(* CoDeSys 2.3.9.41 project: rePlc160.pro *)
(* Libraries: STANDARD.LIB 4.10.05 10:14:46, SmsOwenLib.lib 5.10.12 16:48:36, IECSFC.LIB 13.4.06 14:51:28, Util.lib 18.5.10 15:14:28, SysLibCom.lib 20.2.06 13:31:08, UNM.lib 14.2.06 12:27:08, SMS.lib 29.7.11 08:51:48, SYSLIBTIME.LIB 20.2.06 13:31:16, SYSTASKINFO.LIB 20.2.06 13:31:38, ANALYZATION.LIB 5.10.99 08:05:06, SYSLIBCALLBACK.LIB 20.2.06 13:31:08 *)

(* PLC configuration (modules and I/O channels)
Fast discrete inputs [I_SIMPLE_INPUT] node 0, in %IB0 out %QB0 {Filtrationtime = 10}
  DI_leakSens1 AT %IX0.0 [BitInput] Discrete input 1
  DI_leakSens2 AT %IX0.1 [BitInput] Discrete input 2
  DI_lamp1 AT %IX0.2 [BitInput] Discrete input 3
  DI_lamp2 AT %IX0.3 [BitInput] Discrete input 4
Discrete inputs [ID130] node 1, in %IB1 out %QB1 {Filtrationtime_GeneralINP = 10; Visibility = No; PinCount = 12}
  AT %IB1.0 [ByteInput] DI_POLIW
  AT %IB1.1 [ByteInput] DI_FOUNTAIN
Discrete outputs [ID131] node 2, in %IB2 out %QB2 {SafeValueByte = 0; SafeValueByteM = 0; Visibility = No; PinCount = 12}
  AT %QB2.0 [ByteOutput] DO_POLIW_FOUN_LEAK
  AT %QB2.1 [ByteOutput] DO_FOUN
Fast analog inputs [ID125] node 3, in %IB3 out %QB3 {Flt_Comm = 50Hz 2Por}
  AI_01 AT %IR3.0 [FloatInputP] AI #1 {AIN_TYPE = 0-20 mA; Peak_Filtr = 200; Flt_Ch = Off; TauRC = 10; MinFV = 0; MaxFV = 20000.0}
  AI_02 AT %IR3.1 [FloatInputP] AI #2 {AIN_TYPE = 0-20 mA; Peak_Filtr = 200; Flt_Ch = Off; TauRC = 10; MinFV = 0; MaxFV = 20000.0}
  AI_03 AT %IR3.2 [FloatInputP] AI #3 {AIN_TYPE = 0-20 mA; Peak_Filtr = 200; Flt_Ch = Off; TauRC = 10; MinFV = 0; MaxFV = 20000.0}
  AI_04 AT %IR3.3 [FloatInputP] AI #4 {AIN_TYPE = 0-20 mA; Peak_Filtr = 200; Flt_Ch = Off; TauRC = 10; MinFV = 0; MaxFV = 20000.0}
  AI_05 AT %IR3.4 [FloatInputP] AI #5 {AIN_TYPE = 0-20 mA; Peak_Filtr = 200; Flt_Ch = Off; TauRC = 10; MinFV = 0; MaxFV = 20000.0}
  AI_06 AT %IR3.5 [FloatInputP] AI #6 {AIN_TYPE = 0-20 mA; Peak_Filtr = 200; Flt_Ch = Off; TauRC = 10; MinFV = 0; MaxFV = 20000.0}
  AI_07 AT %IR3.6 [FloatInputP] AI #7 {AIN_TYPE = 0-20 mA; Peak_Filtr = 200; Flt_Ch = Off; TauRC = 10; MinFV = 0; MaxFV = 20000.0}
  AI_08 AT %IR3.7 [FloatInputP] AI #8 {AIN_TYPE = 0-20 mA; Peak_Filtr = 200; Flt_Ch = Off; TauRC = 10; MinFV = 0; MaxFV = 20000.0}
  AT %IW3.8 [WordInput] AI read time (10ms)
Analog outputs [ID126] node 4, in %IB4 out %QB4
  AO_fc AT %QR4.0 [FloatOutputP] AO #1 {AOUT_TYPE = 0-10V; SafeValueREAL = 0.0}
  AO_dim1 AT %QR4.1 [FloatOutputP] AO #2 {AOUT_TYPE = 0-10V; SafeValueREAL = 0.0}
  AO_dim2 AT %QR4.2 [FloatOutputP] AO #3 {AOUT_TYPE = 0-10V; SafeValueREAL = 0.0}
  AO_dim3 AT %QR4.3 [FloatOutputP] AO #4 {AOUT_TYPE = 0-10V; SafeValueREAL = 0.0}
Special input [ID103] node 5, in %IB5 out %QB5 {Filtrationtime = 1000; PinCount = 1; WatchDogPeriod = 400; PollPeriod = 3000; Visibility = No}
  AT %IX5.0 [BitInput] Special input
Special output [ID104] node 6, in %IB6 out %QB6 {Visibility = No; PinCount = 1}
  AT %QX6.0 [BitOutput] Special output
Universal network module [UNM_ID300] node 7, in %IB7 out %QB7 {Visibility = No}
  RS-232 [COM2_USART] node 0, in %IB7.0 out %QB7.0 {CommunicationSpeed = 9600; Parity = NO PARITY CHECK; BitLength = 8 bits; StopLength = One stop bit; InterfaceType = RS232; FrameOriented = ASCII; Timeout = 0; Visibility = No}
AT %QD8.0 [DWordOutput] Last address
AT %QW8.1 [WordOutput] Last error
AT %QB8.0.0 [ByteOutput] Line Status
AT %QB8.0.1 [ByteOutput] Modem Fault
AT %QB8.0.2 [ByteOutput] Start_Auto_Dial
AT %QB8.0.3 [ByteOutput] Stop_Dial
RS-232 [COM2_USART] node 0, in %IB8.0.0 out %QB8.0.0 {CommunicationSpeed = 9600; Parity = NO PARITY CHECK; BitLength = 8 bits; StopLength = One stop bit; InterfaceType = RS232; FrameOriented = ASCII; Timeout = 0; Visibility = No}
PPP_Driver [PPP] node 1, in %IB8.0.1 out %QB8.0.1 {LoginString = mts; PasswordString = mts}
Universal Modbus device [ID2000] node 1, in %IB8.1 out %QB8.1 {ModuleIP = 10:10:122:200; ServiceTimeout = 150; TCPport = 502; NetMode = TCP; ModuleSlaveAddress = 1; RequestType = By command; PeriodOfService = 1000; Visibility = No; RepeatCounter = 0; ByteSequence = Trace_mode}
  AT %QB8.1.0 [ComChannel] Command (0xff - Start)
pad_PoliwDIST AT %IW8.1.0.0 [WordInput]
pad_PoliwTELE AT %QW8.1.1.0 [WordOutput]
Register input module [ID2003] node 2, in %IB8.1.2 out %QB8.1.2 {ModbusAddress = 0; Command_read_regs = Read holding Registers  (0x03); Visibility = No}
  FounDIST AT %IW8.1.2.0 [WordInput]
Register output module [ID2004] node 3, in %IB8.1.3 out %QB8.1.3 {ModbusAddress = 0; Command_write_one_reg = Preset singl register (0x06); Visibility = No}
  FounTELE AT %QW8.1.3.0 [WordOutput]
Register output module [ID2004] node 4, in %IB8.1.4 out %QB8.1.4 {ModbusAddress = 0; Command_write_one_reg = Preset singl register (0x06); Visibility = No}
  TRMOUTS AT %QW8.1.4.0 [WordOutput]
AT %QB8.2.0 [ComChannel] Command (0xff - Start)
pad_Voltage AT %QW8.2.0.0 [WordOutput]
pad_Power_A AT %QW8.2.1.0 [WordOutput]
pad_Power_B AT %QW8.2.2.0 [WordOutput]
pad_Power_C AT %QW8.2.3.0 [WordOutput]
pad_Energy AT %QW8.2.4.0 [WordOutput]
pad_trm1_ch1 AT %QW8.2.5.0 [WordOutput]
pad_trm1_ch2 AT %QW8.2.6.0 [WordOutput]
pad_trm1_set1 AT %QW8.2.7.0 [WordOutput]
pad_trm1_set2 AT %QW8.2.8.0 [WordOutput]
pad_trm2_ch1 AT %QW8.2.9.0 [WordOutput]
pad_trm2_ch2 AT %QW8.2.10.0 [WordOutput]
Register output module [ID2004] node 11, in %IB8.2.11 out %QB8.2.11 {ModbusAddress = 11; Command_write_one_reg = Preset singl register (0x06); Visibility = No}
  pad_trm2_set1 AT %QW8.2.11.0 [WordOutput]
Register output module [ID2004] node 12, in %IB8.2.12 out %QB8.2.12 {ModbusAddress = 12; Command_write_one_reg = Preset singl register (0x06); Visibility = No}
  pad_trm2_set2 AT %QW8.2.12.0 [WordOutput]
Universal Modbus device [ID2000] node 3, in %IB8.3 out %QB8.3 {ModuleIP = 10:10:122:200; ServiceTimeout = 150; TCPport = 502; NetMode = TCP; ModuleSlaveAddress = 1; RequestType = By command; PeriodOfService = 7000; Visibility = No; RepeatCounter = 0; ByteSequence = Trace_mode}
  AT %QB8.3.0 [ComChannel] Command (0xff - Start)
  Register input module [ID2003] node 0, in %IB8.3.0 out %QB8.3.0 {ModbusAddress = 0; Command_read_regs = Read holding Registers  (0x03); Visibility = No}
    cir1On AT %IW8.3.0.0 [WordInput]
  Register input module [ID2003] node 1, in %IB8.3.1 out %QB8.3.1 {ModbusAddress = 0; Command_read_regs = Read holding Registers  (0x03); Visibility = No}
    cir1Off AT %IW8.3.1.0 [WordInput]
  Register input module [ID2003] node 2, in %IB8.3.2 out %QB8.3.2 {ModbusAddress = 0; Command_read_regs = Read holding Registers  (0x03); Visibility = No}
    cir2On AT %IW8.3.2.0 [WordInput]
  Register input module [ID2003] node 3, in %IB8.3.3 out %QB8.3.3 {ModbusAddress = 0; Command_read_regs = Read holding Registers  (0x03); Visibility = No}
    cir2Off AT %IW8.3.3.0 [WordInput]
  Register input module [ID2003] node 4, in %IB8.3.4 out %QB8.3.4 {ModbusAddress = 0; Command_read_regs = Read holding Registers  (0x03); Visibility = No}
    cir3On AT %IW8.3.4.0 [WordInput]
  Register input module [ID2003] node 5, in %IB8.3.5 out %QB8.3.5 {ModbusAddress = 0; Command_read_regs = Read holding Registers  (0x03); Visibility = No}
    cir3Off AT %IW8.3.5.0 [WordInput]
  Register input module [ID2003] node 6, in %IB8.3.6 out %QB8.3.6 {ModbusAddress = 0; Command_read_regs = Read holding Registers  (0x03); Visibility = No}
    dist_staticFValue AT %IW8.3.6.0 [WordInput]
  Register input module [ID2003] node 7, in %IB8.3.7 out %QB8.3.7 {ModbusAddress = 0; Command_read_regs = Read holding Registers  (0x03); Visibility = No}
    p1 AT %IW8.3.7.0 [WordInput]
  Register input module [ID2003] node 8, in %IB8.3.8 out %QB8.3.8 {ModbusAddress = 0; Command_read_regs = Read holding Registers  (0x03); Visibility = No}
    p2 AT %IW8.3.8.0 [WordInput]
  Register input module [ID2003] node 9, in %IB8.3.9 out %QB8.3.9 {ModbusAddress = 0; Command_read_regs = Read holding Registers  (0x03); Visibility = No}
    p3 AT %IW8.3.9.0 [WordInput]
  Register input module [ID2003] node 10, in %IB8.3.10 out %QB8.3.10 {ModbusAddress = 0; Command_read_regs = Read holding Registers  (0x03); Visibility = No}
    p4 AT %IW8.3.10.0 [WordInput]
  Register input module [ID2003] node 11, in %IB8.3.11 out %QB8.3.11 {ModbusAddress = 0; Command_read_regs = Read holding Registers  (0x03); Visibility = No}
    p5 AT %IW8.3.11.0 [WordInput]
  Register input module [ID2003] node 12, in %IB8.3.12 out %QB8.3.12 {ModbusAddress = 0; Command_read_regs = Read holding Registers  (0x03); Visibility = No}
    p6 AT %IW8.3.12.0 [WordInput]
  Register input module [ID2003] node 13, in %IB8.3.13 out %QB8.3.13 {ModbusAddress = 0; Command_read_regs = Read holding Registers  (0x03); Visibility = No}
    p7 AT %IW8.3.13.0 [WordInput]
  Register input module [ID2003] node 14, in %IB8.3.14 out %QB8.3.14 {ModbusAddress = 0; Command_read_regs = Read holding Registers  (0x03); Visibility = No}
    p8 AT %IW8.3.14.0 [WordInput]
  Register input module [ID2003] node 15, in %IB8.3.15 out %QB8.3.15 {ModbusAddress = 0; Command_read_regs = Read holding Registers  (0x03); Visibility = No}
    p9 AT %IW8.3.15.0 [WordInput]
  Register input module [ID2003] node 16, in %IB8.3.16 out %QB8.3.16 {ModbusAddress = 0; Command_read_regs = Read holding Registers  (0x03); Visibility = No}
    p10 AT %IW8.3.16.0 [WordInput]
  Register input module [ID2003] node 17, in %IB8.3.17 out %QB8.3.17 {ModbusAddress = 0; Command_read_regs = Read holding Registers  (0x03); Visibility = No}
    trm1_ch1_day AT %IW8.3.17.0 [WordInput]
  Register input module [ID2003] node 18, in %IB8.3.18 out %QB8.3.18 {ModbusAddress = 0; Command_read_regs = Read holding Registers  (0x03); Visibility = No}
    trm1_ch1_night AT %IW8.3.18.0 [WordInput]
  Register input module [ID2003] node 19, in %IB8.3.19 out %QB8.3.19 {ModbusAddress = 0; Command_read_regs = Read holding Registers  (0x03); Visibility = No}
    trm1_ch2_day AT %IW8.3.19.0 [WordInput]
  Register input module [ID2003] node 20, in %IB8.3.20 out %QB8.3.20 {ModbusAddress = 0; Command_read_regs = Read holding Registers  (0x03); Visibility = No}
    trm1_ch2_night AT %IW8.3.20.0 [WordInput]
  Register input module [ID2003] node 21, in %IB8.3.21 out %QB8.3.21 {ModbusAddress = 0; Command_read_regs = Read holding Registers  (0x03); Visibility = No}
    trm2_ch1_day AT %IW8.3.21.0 [WordInput]
  Register input module [ID2003] node 22, in %IB8.3.22 out %QB8.3.22 {ModbusAddress = 0; Command_read_regs = Read holding Registers  (0x03); Visibility = No}
    trm2_ch1_night AT %IW8.3.22.0 [WordInput]
  Register input module [ID2003] node 23, in %IB8.3.23 out %QB8.3.23 {ModbusAddress = 0; Command_read_regs = Read holding Registers  (0x03); Visibility = No}
    trm2_ch2_day AT %IW8.3.23.0 [WordInput]
  Register input module [ID2003] node 24, in %IB8.3.24 out %QB8.3.24 {ModbusAddress = 0; Command_read_regs = Read holding Registers  (0x03); Visibility = No}
    trm2_ch2_night AT %IW8.3.24.0 [WordInput]
  Register input module [ID2003] node 25, in %IB8.3.25 out %QB8.3.25 {ModbusAddress = 0; Command_read_regs = Read holding Registers  (0x03); Visibility = No}
    trm1_ch1_dayVal AT %IW8.3.25.0 [WordInput]
  Register input module [ID2003] node 26, in %IB8.3.26 out %QB8.3.26 {ModbusAddress = 0; Command_read_regs = Read holding Registers  (0x03); Visibility = No}
    trm1_ch1_nightVal AT %IW8.3.26.0 [WordInput]
  Register input module [ID2003] node 27, in %IB8.3.27 out %QB8.3.27 {ModbusAddress = 0; Command_read_regs = Read holding Registers  (0x03); Visibility = No}
    trm1_ch2_dayVal AT %IW8.3.27.0 [WordInput]
  Register input module [ID2003] node 28, in %IB8.3.28 out %QB8.3.28 {ModbusAddress = 0; Command_read_regs = Read holding Registers  (0x03); Visibility = No}
    trm1_ch2_nightVal AT %IW8.3.28.0 [WordInput]
  Register input module [ID2003] node 29, in %IB8.3.29 out %QB8.3.29 {ModbusAddress = 0; Command_read_regs = Read holding Registers  (0x03); Visibility = No}
    trm2_ch1_dayVal AT %IW8.3.29.0 [WordInput]
  Register input module [ID2003] node 30, in %IB8.3.30 out %QB8.3.30 {ModbusAddress = 0; Command_read_regs = Read holding Registers  (0x03); Visibility = No}
    trm2_ch1_nightVal AT %IW8.3.30.0 [WordInput]
  Register input module [ID2003] node 31, in %IB8.3.31 out %QB8.3.31 {ModbusAddress = 0; Command_read_regs = Read holding Registers  (0x03); Visibility = No}
    trm2_ch2_dayVal AT %IW8.3.31.0 [WordInput]
  Register input module [ID2003] node 32, in %IB8.3.32 out %QB8.3.32 {ModbusAddress = 0; Command_read_regs = Read holding Registers  (0x03); Visibility = No}
    trm2_ch2_nightVal AT %IW8.3.32.0 [WordInput]
ModBus (slave) [MODBUS_ID400] node 9, in %IB9 out %QB9 {SlaveIdentificator = 1; Visibility = No}
  Modbus [MODBUS_ID302] node 0, in %IB9.0 out %QB9.0
    TCP [TCP_ID221] node 0, in %IB9.0.0 out %QB9.0.0 {RemotePort = 502; Visibility = No}
  2 byte [Register] node 1, in %IB9.1 out %QB9.1
    dim1 AT %QW9.1.0 [WordOutput]
  2 byte [Register] node 2, in %IB9.2 out %QB9.2
    dim2 AT %QW9.2.0 [WordOutput]
  2 byte [Register] node 3, in %IB9.3 out %QB9.3
    dim3 AT %QW9.3.0 [WordOutput]
  2 byte [Register] node 4, in %IB9.4 out %QB9.4
    weBITS_IN AT %QW9.4.0 [WordOutput] (leak)
  2 byte [Register] node 5, in %IB9.5 out %QB9.5
    weBITS_OUT AT %QW9.5.0 [WordOutput] leakSens1,leakSens2,valveStat,drePumpStat,unknPump
  2 byte [Register] node 6, in %IB9.6 out %QB9.6
    AI1_OUT AT %QW9.6.0 [WordOutput]
  2 byte [Register] node 7, in %IB9.7 out %QB9.7
    AI2_OUT AT %QW9.7.0 [WordOutput]
  2 byte [Register] node 8, in %IB9.8 out %QB9.8
    AI3_OUT AT %QW9.8.0 [WordOutput]
  2 byte [Register] node 9, in %IB9.9 out %QB9.9
    AI4_OUT AT %QW9.9.0 [WordOutput]
  2 byte [Register] node 10, in %IB9.10 out %QB9.10
    AI5_OUT AT %QW9.10.0 [WordOutput]
  2 byte [Register] node 11, in %IB9.11 out %QB9.11
    AI6_OUT AT %QW9.11.0 [WordOutput]
  2 byte [Register] node 12, in %IB9.12 out %QB9.12
    AI7_OUT AT %QW9.12.0 [WordOutput]
  2 byte [Register] node 13, in %IB9.13 out %QB9.13
    AI8_OUT AT %QW9.13.0 [WordOutput]
  2 byte [Register] node 14, in %IB9.14 out %QB9.14
    DrenageBITS AT %QW9.14.0 [WordOutput]
  2 byte [Register] node 15, in %IB9.15 out %QB9.15
    dist_top AT %QW9.15.0 [WordOutput]
  2 byte [Register] node 16, in %IB9.16 out %QB9.16
    dist_bottom AT %QW9.16.0 [WordOutput]
  2 byte [Register] node 17, in %IB9.17 out %QB9.17
    sens4ma AT %QW9.17.0 [WordOutput]
  2 byte [Register] node 18, in %IB9.18 out %QB9.18
    sens20ma AT %QW9.18.0 [WordOutput]
  2 byte [Register] node 19, in %IB9.19 out %QB9.19
    dist_LAMP AT %QW9.19.0 [WordOutput]
  2 byte [Register] node 20, in %IB9.20 out %QB9.20
    tele_LAMP AT %QW9.20.0 [WordOutput]
  2 byte [Register] node 21, in %IB9.21 out %QB9.21
    lamp1On AT %QW9.21.0 [WordOutput]
  2 byte [Register] node 22, in %IB9.22 out %QB9.22
    lamp1Off AT %QW9.22.0 [WordOutput]
  2 byte [Register] node 23, in %IB9.23 out %QB9.23
    lamp2On AT %QW9.23.0 [WordOutput]
  2 byte [Register] node 24, in %IB9.24 out %QB9.24
    lamp2Off AT %QW9.24.0 [WordOutput]
  2 byte [Register] node 25, in %IB9.25 out %QB9.25
    lamp3On AT %QW9.25.0 [WordOutput]
  2 byte [Register] node 26, in %IB9.26 out %QB9.26
    lamp3Off AT %QW9.26.0 [WordOutput]
  2 byte [Register] node 27, in %IB9.27 out %QB9.27
    dreOUT AT %QW9.27.0 [WordOutput]
  2 byte [Register] node 28, in %IB9.28 out %QB9.28
    someDIs AT %QW9.28.0 [WordOutput]
  2 byte [Register] node 29, in %IB9.29 out %QB9.29
    door AT %QW9.29.0 [WordOutput]
  2 byte [Register] node 30, in %IB9.30 out %QB9.30
    year AT %QW9.30.0 [WordOutput]
  2 byte [Register] node 31, in %IB9.31 out %QB9.31
    monthday AT %QW9.31.0 [WordOutput]
  2 byte [Register] node 32, in %IB9.32 out %QB9.32
    hourminute AT %QW9.32.0 [WordOutput]
  2 byte [Register] node 33, in %IB9.33 out %QB9.33
    tele_year AT %QW9.33.0 [WordOutput]
  2 byte [Register] node 34, in %IB9.34 out %QB9.34
    tele_month AT %QW9.34.0 [WordOutput]
  2 byte [Register] node 35, in %IB9.35 out %QB9.35
    tele_day AT %QW9.35.0 [WordOutput]
  2 byte [Register] node 36, in %IB9.36 out %QB9.36
    tele_hour AT %QW9.36.0 [WordOutput]
  2 byte [Register] node 37, in %IB9.37 out %QB9.37
    tele_minute AT %QW9.37.0 [WordOutput]
  2 byte [Register] node 38, in %IB9.38 out %QB9.38
    door_delay AT %QW9.38.0 [WordOutput]
  2 byte [Register] node 39, in %IB9.39 out %QB9.39
    transfer_di AT %QW9.39.0 [WordOutput]
  2 byte [Register] node 40, in %IB9.40 out %QB9.40
    transfer_do AT %QW9.40.0 [WordOutput]
ModBus (Master) [MODBUS_MASTER_ID450] node 10, in %IB10 out %QB10 {Visibility = No}
  AT %QD10.0 [DWordOutput] Last address
  AT %QW10.1 [WordOutput] Last error
  RS-485-1 [COM1_USART] node 0, in %IB10.0 out %QB10.0 {CommunicationSpeed = 19200; Parity = NO PARITY CHECK; BitLength = 8 bits; StopLength = Two stop bits; InterfaceType = RS485; FrameOriented = RTU; Timeout = 0; Visibility = No}
  Universal Modbus device [ID2000] node 1, in %IB10.1 out %QB10.1 {ModuleIP = 10:0:0:223; ServiceTimeout = 150; TCPport = 502; NetMode = Serial; ModuleSlaveAddress = 4; RequestType = By poll time; PeriodOfService = 5000; Visibility = No; RepeatCounter = 0; ByteSequence = Trace_mode}
    AT %QB10.1.0 [ComChannel] Command (0xff - Start)
    32bit input module [ID2005] node 0, in %IB10.1.0 out %QB10.1.0 {ModbusAddress = 0; Command_read_regs = Read holding Registers  (0x03); Visibility = No}
      Voltage AT %ID10.1.0.0 [DWordInput]
    32bit input module [ID2005] node 1, in %IB10.1.1 out %QB10.1.1 {ModbusAddress = 4; Command_read_regs = Read holding Registers  (0x03); Visibility = No}
      Power_A AT %ID10.1.1.0 [DWordInput]
      Power_B AT %ID10.1.2.0 [DWordInput]
      Power_C AT %ID10.1.3.0 [DWordInput]
      Energy AT %ID10.1.4.0 [DWordInput]
  Universal Modbus device [ID2000] node 2, in %IB10.2 out %QB10.2 {ModuleIP = 10:0:0:223; ServiceTimeout = 150; TCPport = 502; NetMode = Serial; ModuleSlaveAddress = 5; RequestType = By poll time; PeriodOfService = 2000; Visibility = No; RepeatCounter = 0; ByteSequence = Trace_mode}
    AT %QB10.2.0 [ComChannel] Command (0xff - Start)
trm1_ch1 AT %IW10.2.0.0 [WordInput]
trm1_ch2 AT %IW10.2.1.0 [WordInput]
trm1_set1_read AT %IW10.2.2.0 [WordInput]
trm1_set2_read AT %IW10.2.3.0 [WordInput]
trm1_out1 AT %IW10.2.4.0 [WordInput]
trm1_out2 AT %IW10.2.5.0 [WordInput]
Universal Modbus device [ID2000] node 3, in %IB10.3 out %QB10.3 {ModuleIP = 10:0:0:223; ServiceTimeout = 150; TCPport = 502; NetMode = Serial; ModuleSlaveAddress = 5; RequestType = By value change; PeriodOfService = 10000; Visibility = No; RepeatCounter = 0; ByteSequence = Trace_mode}
  AT %QB10.3.0 [ComChannel] Command (0xff - Start)
trm1_set1_write AT %QW10.3.0.0 [WordOutput]
trm1_set2_write AT %QW10.3.1.0 [WordOutput]
Universal Modbus device [ID2000] node 4, in %IB10.4 out %QB10.4 {ModuleIP = 10:0:0:223; ServiceTimeout = 150; TCPport = 502; NetMode = Serial; ModuleSlaveAddress = 6; RequestType = By poll time; PeriodOfService = 2000; Visibility = No; RepeatCounter = 0; ByteSequence = Trace_mode}
  AT %QB10.4.0 [ComChannel] Command (0xff - Start)
trm2_ch1 AT %IW10.4.0.0 [WordInput]
trm2_ch2 AT %IW10.4.1.0 [WordInput]
trm2_set1_read AT %IW10.4.2.0 [WordInput]
trm2_set2_read AT %IW10.4.3.0 [WordInput]
trm2_out1 AT %IW10.4.4.0 [WordInput]
trm2_out2 AT %IW10.4.5.0 [WordInput]
Universal Modbus device [ID2000] node 5, in %IB10.5 out %QB10.5 {ModuleIP = 10:0:0:223; ServiceTimeout = 150; TCPport = 502; NetMode = Serial; ModuleSlaveAddress = 6; RequestType = By value change; PeriodOfService = 10000; Visibility = No; RepeatCounter = 0; ByteSequence = Trace_mode}
  AT %QB10.5.0 [ComChannel] Command (0xff - Start)
trm2_set1_write AT %QW10.5.0.0 [WordOutput]
trm2_set2_write AT %QW10.5.1.0 [WordOutput]
*)

(* Global variable list: Global_Variables *)
VAR_GLOBAL

(* Times *)
	GetTime: CurTimeEx;
	TimeAndDate: SystemTimeDate;
	Sys_Time: SysTime64;

	SMS_ID  : WORD;

	DI_door : BOOL := FALSE;
	DO_door : BOOL := FALSE;
	DO_drePump : BOOL := FALSE;
	DO_unknownPump : BOOL := FALSE;
	DI_staticMode : BOOL := FALSE;
	DI_dynamicMode : BOOL := FALSE;
	DI_v1_manMode : BOOL := FALSE;
	DI_v2_manMode : BOOL := FALSE;
	DI_v3_manMode : BOOL := FALSE;
	DO_pump : BOOL := FALSE;
	DI_pumpState : BOOL := FALSE;

END_VAR

(* POU PLC_PRG, ST *)
PROGRAM PLC_PRG
VAR
	NO_FIRST_PASS : BOOL;
	FP_door1: R_TRIG;
	i_change: BOOL;
	dorr_timer: TON;
	door_time : TIME;
END_VAR
VAR RETAIN
	weBITS_IN_save : WORD;
END_VAR
(*
закомменчены:
FOUNTAIN WithdrawRetain
POLIW WithdrawRetain
TRM WithdrawRetain
*)
IF NO_FIRST_PASS = FALSE
	THEN _WithdrawRetain;
	NO_FIRST_PASS := TRUE;
END_IF;

_CheckNewValue;

_Leakage;

door_time := WORD_TO_TIME ( door_delay );
_Door;

_Tele;

POLIW;

FOUNTAIN;

TRM;

_CVM;

LIGHT;

DRENAGE;

SMS;
END_PROGRAM
ACTION _CheckNewValue:
IF weBITS_IN_save <> weBITS_IN
	THEN weBITS_IN_save := weBITS_IN;
END_IF;
END_ACTION
ACTION _CVM:
pad_Voltage := DWORD_TO_WORD( Voltage );
pad_Power_A := DWORD_TO_WORD( Power_A );
pad_Power_B := DWORD_TO_WORD( Power_B );
pad_Power_C := DWORD_TO_WORD( Power_C );
pad_Energy := DWORD_TO_WORD( Energy );
END_ACTION
ACTION _Door:
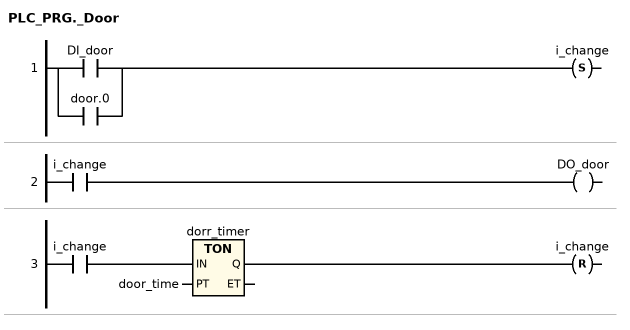
_LD_ (* Ladder Diagram *)
NETWORK 1
	{ [DI_door] | [door.0] } --- (S i_change)
NETWORK 2
	[i_change] --- (DO_door)
NETWORK 3
	[i_change] - dorr_timer:TON(IN: *, PT: door_time) --- (R i_change)
_END_LD_
(* the same logic as Structured Text *)
(* Network 1 *)
IF DI_door OR door.0 THEN i_change := TRUE; END_IF;
(* Network 2 *)
DO_door := i_change;
(* Network 3 *)
dorr_timer(IN := i_change, PT := door_time);
IF dorr_timer.Q THEN i_change := FALSE; END_IF;
END_ACTION
ACTION _Leakage:
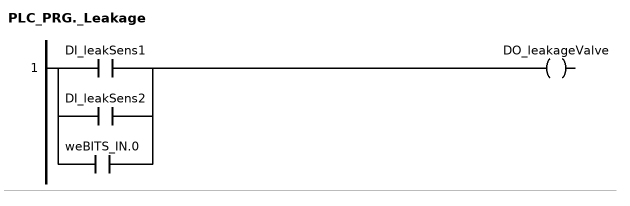
_LD_ (* Ladder Diagram *)
NETWORK 1
	{ [DI_leakSens1] | [DI_leakSens2] | [weBITS_IN.0] } --- (DO_leakageValve)
_END_LD_
(* the same logic as Structured Text *)
(* Network 1 *)
DO_leakageValve := DI_leakSens1 OR DI_leakSens2 OR weBITS_IN.0;
END_ACTION
ACTION _Tele:
weBITS_OUT.0 := DI_leakSens1;
weBITS_OUT.1 := DI_leakSens2;
weBITS_OUT.2 := DO_leakageValve;

AI1_OUT := REAL_TO_WORD ( AI_01 );
AI2_OUT := REAL_TO_WORD ( AI_02 );
AI3_OUT := REAL_TO_WORD ( AI_03 );
AI4_OUT := REAL_TO_WORD ( AI_04 );
AI5_OUT := REAL_TO_WORD ( AI_05 );
AI6_OUT := REAL_TO_WORD ( AI_06 );
AI7_OUT := REAL_TO_WORD ( AI_07 );
AI8_OUT := REAL_TO_WORD ( AI_08 );
(*
someDIs.0 := DI_konduk;*)
someDIs.1 := DI_powerSupply;(*
someDIs.2 := DI_banya;
someDIs.3 := DI_pool;
someDIs.4 := DI_foun;
someDIs.5 := DI_poliw;
someDIs.6 := DO_door;*)

transfer_di.0 := DI_leakSens1;
transfer_di.1 := DI_leakSens2;
transfer_di.2 := DI_lamp1;
transfer_di.3 := DI_lamp2;
transfer_di.4 := DI_lamp3;
transfer_di.5 := DI_rainSens;
transfer_di.6 := DI_powerSupply;
transfer_di.7 := DI_signal1;
transfer_di.8 := DI_signal2;
transfer_di.9 := DI_fireSignal;(*
transfer_di.10 :=
transfer_di.11 := DI_banya;
transfer_di.12 := DI_staticMode;
transfer_di.13 := DI_dynamicMode;
transfer_di.14 :=
transfer_di.15 := DI_pool;*)

transfer_do.0 := DO_valve1;
transfer_do.1 := DO_valve2;
transfer_do.2 := DO_valve3;
(*transfer_do.3 := DO_pump;*)
transfer_do.4 := DO_founPump;
transfer_do.5 := DO_leakageValve;
transfer_do.6 := DO_door;
transfer_do.7 := DO_unknownPump;
transfer_do.8 := DO_drePump;
transfer_do.9 := DO_lamp1;
transfer_do.10 := DO_lamp2;
transfer_do.11 := DO_lamp3;
END_ACTION
ACTION _WithdrawRetain:
weBITS_IN := weBITS_IN_save;
END_ACTION

(* POU POLIW, ST *)
PROGRAM POLIW
VAR
	NO_FIRST_PASS : BOOL;
	PUNCH : WORD;
	setYear : INT;
	setMonth, setDay, setHour, setMinute : BYTE;
	set_time : BOOL;

(* bits *)
	dist_valve1, dist_valve2, dist_valve3, dist_valve4, dist_exMech : BOOL;

	dist_manka : BOOL;

	MON : BOOL;
	TUE : BOOL;
	WED : BOOL;
	THU : BOOL;
	FRI : BOOL;
	SAT : BOOL;
	SUN : BOOL;

	cir1OnHH, cir1OnMM, cir1OffHH, cir1OffMM,
	cir2OnHH, cir2OnMM, cir2OffHH, cir2OffMM,
	cir3OnHH, cir3OnMM, cir3OffHH, cir3OffMM,
	cir4OnHH, cir4OnMM, cir4OffHH, cir4OffMM : BYTE;


	tele_pumpState, tele_v1state, tele_v2state, tele_v3state, tele_v4state, tele_exMechState,
	tele_rainSens, tele_humSens : BOOL;

	cir1mustRun: BOOL;
	cir2mustRun: BOOL;
	cir3mustRun: BOOL;
	cir4mustRun: BOOL;
	dayOk: BOOL;

	isGalet234 : BOOL;

	waterFault: BOOL;

	auto_pump_start: BOOL;
	auto_v1_open: BOOL;
	auto_v2_open: BOOL;
	auto_v3_open: BOOL;
	auto_v4_open : BOOL;

	dist_pump_start: BOOL;
	dist_v1_open: BOOL;
	dist_v2_open: BOOL;
	dist_v3_open: BOOL;
	dist_v4_open: BOOL;

	v1_auto_started: BOOL;
	FN_dist_v1_off: F_TRIG;
	v1_must_dist_stop: BOOL;
	v2_auto_started: BOOL;
	FN_dist_v2_off: F_TRIG;
	v2_must_dist_stop: BOOL;
	v3_auto_started: BOOL;
	FN_dist_v3_off: F_TRIG;
	v3_must_dist_stop: BOOL;
END_VAR

VAR RETAIN

	SAVE_BITS : WORD;

	save_cir1On, save_cir1Off, save_cir2On, save_cir2Off,
	save_cir3On, save_cir3Off, save_cir4On, save_cir4Off : WORD;

	save_year, save_monthday, save_hourminute : WORD;
END_VAR
(* 				first pass 				*)
IF NO_FIRST_PASS = FALSE
	THEN WithdrawRetain;
	PUNCH := 65535;
	Obtaining;
	PUNCH := 0;
	NO_FIRST_PASS := TRUE;
END_IF;

(*			    main cycle		  		*)
PUNCH := 0;

set_time := door.1;
Times; (* получение текущего времени *)

CheckNewVal; (* проверка наличия новых значений переменных из модбас *)
				 (* и запись их в retain переменные *)
IF PUNCH > 0 THEN
	Obtaining; (* распаковка retain переменных в рабочие переменные *)
END_IF;

Schedule; (* основной цикл полива *)
(*
ExMech; (* управление исполнительным механизмом *)
*)
Outs; (* управление выходами контроллера на полив *)

HandOff;
Tele; (* передача рабочего состояния на верхний уровень *)
END_PROGRAM
ACTION CheckNewVal:
IF SAVE_BITS <> pad_PoliwDIST
	THEN SAVE_BITS := pad_PoliwDIST;
			PUNCH.0 := TRUE;
END_IF;



IF save_cir1On <> cir1On
	THEN save_cir1On := cir1On;
			PUNCH.1 := TRUE;
END_IF;

IF save_cir1Off <> cir1Off
	THEN save_cir1Off := cir1Off;
			PUNCH.2 := TRUE;
END_IF;


IF save_cir2On <> cir2On
	THEN save_cir2On := cir2On;
			PUNCH.3 := TRUE;
END_IF;

IF save_cir2Off <> cir2Off
	THEN save_cir2Off := cir2Off;
			PUNCH.4 := TRUE;
END_IF;


IF save_cir3On <> cir3On
	THEN save_cir3On := cir3On;
			PUNCH.5 := TRUE;
END_IF;

IF save_cir3Off <> cir3Off
	THEN save_cir3Off := cir3Off;
			PUNCH.6 := TRUE;
END_IF;


IF save_year <> year
	THEN save_year := year;
			PUNCH.9 := TRUE;
END_IF;

IF save_monthday <> monthday
	THEN save_monthday := monthday;
			PUNCH.10 := TRUE;
END_IF;

IF save_hourminute <> hourminute
	THEN save_hourminute := hourminute;
			PUNCH.11 := TRUE;
END_IF;
END_ACTION
ACTION HandOff:
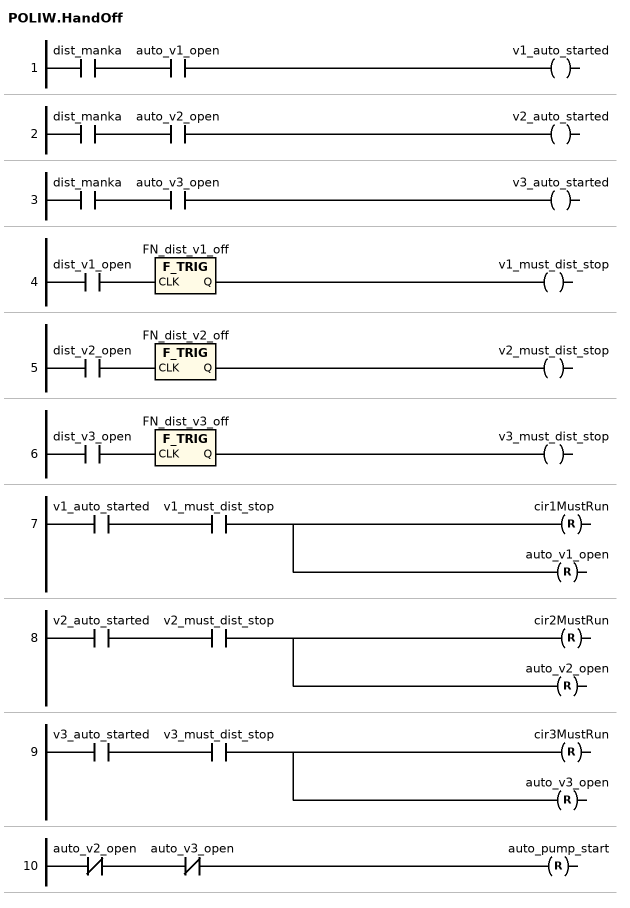
_LD_ (* Ladder Diagram *)
NETWORK 1
	[dist_manka] - [auto_v1_open] --- (v1_auto_started)
NETWORK 2
	[dist_manka] - [auto_v2_open] --- (v2_auto_started)
NETWORK 3
	[dist_manka] - [auto_v3_open] --- (v3_auto_started)
NETWORK 4
	[dist_v1_open] - FN_dist_v1_off:F_TRIG(CLK: *) --- (v1_must_dist_stop)
NETWORK 5
	[dist_v2_open] - FN_dist_v2_off:F_TRIG(CLK: *) --- (v2_must_dist_stop)
NETWORK 6
	[dist_v3_open] - FN_dist_v3_off:F_TRIG(CLK: *) --- (v3_must_dist_stop)
NETWORK 7
	[v1_auto_started] - [v1_must_dist_stop] --- (R cir1MustRun) (R auto_v1_open)
NETWORK 8
	[v2_auto_started] - [v2_must_dist_stop] --- (R cir2MustRun) (R auto_v2_open)
NETWORK 9
	[v3_auto_started] - [v3_must_dist_stop] --- (R cir3MustRun) (R auto_v3_open)
NETWORK 10
	[/auto_v2_open] - [/auto_v3_open] --- (R auto_pump_start)
_END_LD_
(* the same logic as Structured Text *)
(* Network 1 *)
v1_auto_started := dist_manka AND auto_v1_open;
(* Network 2 *)
v2_auto_started := dist_manka AND auto_v2_open;
(* Network 3 *)
v3_auto_started := dist_manka AND auto_v3_open;
(* Network 4 *)
FN_dist_v1_off(CLK := dist_v1_open);
v1_must_dist_stop := FN_dist_v1_off.Q;
(* Network 5 *)
FN_dist_v2_off(CLK := dist_v2_open);
v2_must_dist_stop := FN_dist_v2_off.Q;
(* Network 6 *)
FN_dist_v3_off(CLK := dist_v3_open);
v3_must_dist_stop := FN_dist_v3_off.Q;
(* Network 7 *)
IF v1_auto_started AND v1_must_dist_stop THEN cir1MustRun := FALSE; auto_v1_open := FALSE; END_IF;
(* Network 8 *)
IF v2_auto_started AND v2_must_dist_stop THEN cir2MustRun := FALSE; auto_v2_open := FALSE; END_IF;
(* Network 9 *)
IF v3_auto_started AND v3_must_dist_stop THEN cir3MustRun := FALSE; auto_v3_open := FALSE; END_IF;
(* Network 10 *)
IF NOT auto_v2_open AND NOT auto_v3_open THEN auto_pump_start := FALSE; END_IF;
END_ACTION
ACTION Obtaining:
IF PUNCH.0 THEN
	dist_manka := SAVE_BITS.0;
	dist_valve1 := SAVE_BITS.1;
	dist_valve2 := SAVE_BITS.2;
	dist_valve3 := SAVE_BITS.3;
	dist_valve4 := SAVE_BITS.4;
	dist_exMech := SAVE_BITS.5;

	MON := SAVE_BITS.6;
	TUE := SAVE_BITS.7;
	WED := SAVE_BITS.8;
	THU := SAVE_BITS.9;
	FRI := SAVE_BITS.10;
	SAT := SAVE_BITS.11;
	SUN := SAVE_BITS.12;

	PUNCH.0 := FALSE;
END_IF;

(*
	lo,hi : byte
	w : word

	lo := word_to_byte(w)
	hi := word_to_byte(w/256)
	w := 256*hi + lo 
*)

IF PUNCH.1 THEN
	cir1OnHH := WORD_TO_BYTE ( save_cir1On );
	cir1OnMM := WORD_TO_BYTE ( save_cir1On / 256 );
	PUNCH.1 := FALSE;
END_IF;

IF PUNCH.2 THEN
	cir1OffHH := WORD_TO_BYTE ( save_cir1Off );
	cir1OffMM := WORD_TO_BYTE ( save_cir1Off / 256 );
	PUNCH.2 := FALSE;
END_IF;

IF PUNCH.3 THEN
	cir2OnHH := WORD_TO_BYTE ( save_cir2On );
	cir2OnMM := WORD_TO_BYTE ( save_cir2On / 256 );
	PUNCH.3 := FALSE;
END_IF;

IF PUNCH.4 THEN
	cir2OffHH := WORD_TO_BYTE ( save_cir2Off );
	cir2OffMM := WORD_TO_BYTE ( save_cir2Off / 256 );
	PUNCH.4 := FALSE;
END_IF;

IF PUNCH.5 THEN
	cir3OnHH := WORD_TO_BYTE ( save_cir3On );
	cir3OnMM := WORD_TO_BYTE ( save_cir3On / 256 );
	PUNCH.5 := FALSE;
END_IF;

IF PUNCH.6 THEN
	cir3OffHH := WORD_TO_BYTE ( save_cir3Off );
	cir3OffMM := WORD_TO_BYTE ( save_cir3Off / 256 );
	PUNCH.6 := FALSE;
END_IF;

IF PUNCH.7 THEN
	cir4OnHH := WORD_TO_BYTE ( save_cir4On );
	cir4OnMM := WORD_TO_BYTE ( save_cir4On / 256 );
	PUNCH.7 := FALSE;
END_IF;

IF PUNCH.8 THEN
	cir4OffHH := WORD_TO_BYTE ( save_cir4Off );
	cir4OffMM := WORD_TO_BYTE ( save_cir4Off / 256 );
	PUNCH.8 := FALSE;
END_IF;

IF PUNCH.9 THEN
	setYear := WORD_TO_INT ( save_year );
	PUNCH.9 := FALSE;
END_IF;

IF PUNCH.10 THEN
	setDay := WORD_TO_BYTE ( save_monthday );
	setMonth := WORD_TO_BYTE ( save_monthday / 256 );
	PUNCH.10 := FALSE;
END_IF;

IF PUNCH.11 THEN
	setMinute := WORD_TO_BYTE ( save_hourminute );
	setHour := WORD_TO_BYTE ( save_hourminute / 256 );
	PUNCH.11 := FALSE;
END_IF;
END_ACTION
ACTION Outs:
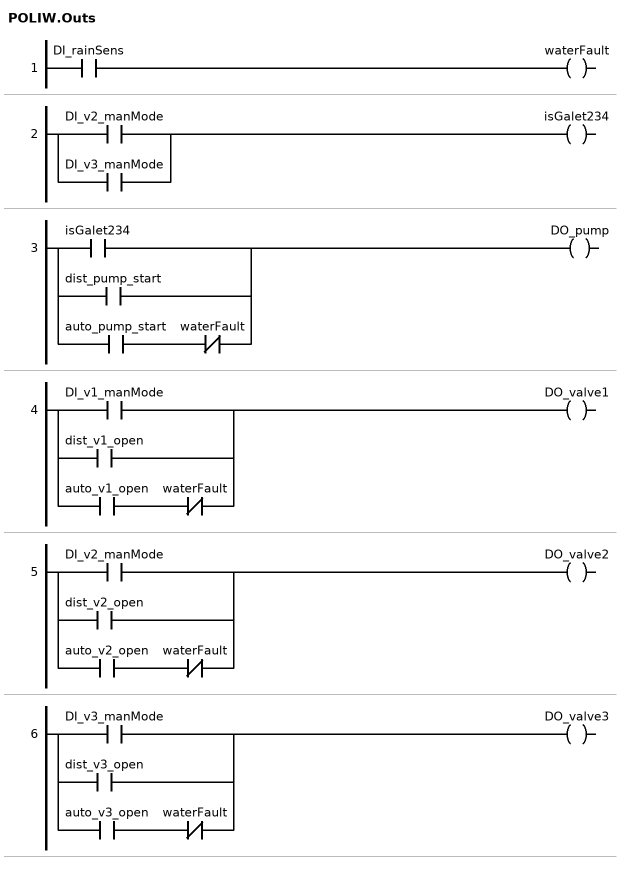
_LD_ (* Ladder Diagram *)
NETWORK 1
	[DI_rainSens] --- (waterFault)
NETWORK 2
	{ [DI_v2_manMode] | [DI_v3_manMode] } --- (isGalet234)
NETWORK 3
	{ [isGalet234] | [dist_pump_start] | [auto_pump_start] - [/waterFault] } --- (DO_pump)
NETWORK 4
	{ [DI_v1_manMode] | [dist_v1_open] | [auto_v1_open] - [/waterFault] } --- (DO_valve1)
NETWORK 5
	{ [DI_v2_manMode] | [dist_v2_open] | [auto_v2_open] - [/waterFault] } --- (DO_valve2)
NETWORK 6
	{ [DI_v3_manMode] | [dist_v3_open] | [auto_v3_open] - [/waterFault] } --- (DO_valve3)
_END_LD_
(* the same logic as Structured Text *)
(* Network 1 *)
waterFault := DI_rainSens;
(* Network 2 *)
isGalet234 := DI_v2_manMode OR DI_v3_manMode;
(* Network 3 *)
DO_pump := isGalet234 OR dist_pump_start OR auto_pump_start AND NOT waterFault;
(* Network 4 *)
DO_valve1 := DI_v1_manMode OR dist_v1_open OR auto_v1_open AND NOT waterFault;
(* Network 5 *)
DO_valve2 := DI_v2_manMode OR dist_v2_open OR auto_v2_open AND NOT waterFault;
(* Network 6 *)
DO_valve3 := DI_v3_manMode OR dist_v3_open OR auto_v3_open AND NOT waterFault;
END_ACTION
ACTION Schedule:
(* контур 1 *)
IF ( cir1OnHH = TimeAndDate.Hour ) AND ( cir1OnMM = TimeAndDate.Minute ) AND ( TimeAndDate.Second = 0 )
	THEN cir1mustRun := TRUE;
END_IF;

IF ( cir1OffHH = TimeAndDate.Hour ) AND ( cir1OffMM = TimeAndDate.Minute ) AND ( TimeAndDate.Second = 0 )
	THEN cir1mustRun := FALSE;
END_IF;

(* контур 2 *)
IF ( cir2OnHH = TimeAndDate.Hour ) AND ( cir2OnMM = TimeAndDate.Minute ) AND ( TimeAndDate.Second = 0 )
	THEN cir2mustRun := TRUE;
END_IF;

IF ( cir2OffHH = TimeAndDate.Hour ) AND ( cir2OffMM = TimeAndDate.Minute ) AND ( TimeAndDate.Second = 0 )
	THEN cir2mustRun := FALSE;
END_IF;

(* контур 3 *)
IF ( cir3OnHH = TimeAndDate.Hour ) AND ( cir3OnMM = TimeAndDate.Minute ) AND ( TimeAndDate.Second = 0 )
	THEN cir3mustRun := TRUE;
END_IF;

IF ( cir3OffHH = TimeAndDate.Hour ) AND ( cir3OffMM = TimeAndDate.Minute ) AND ( TimeAndDate.Second = 0 )
	THEN cir3mustRun := FALSE;
END_IF;

(* контур 4 *)
IF ( cir4OnHH = TimeAndDate.Hour ) AND ( cir4OnMM = TimeAndDate.Minute ) AND ( TimeAndDate.Second = 0 )
	THEN cir4mustRun := TRUE;
END_IF;

IF ( cir4OffHH = TimeAndDate.Hour ) AND ( cir4OffMM = TimeAndDate.Minute ) AND ( TimeAndDate.Second = 0 )
	THEN cir4mustRun := FALSE;
END_IF;

(* день недели *)
CASE TimeAndDate.DayOfWeek OF
	1 : IF MON
	     	THEN dayOk := TRUE;
		ELSE dayOk := FALSE;
	     END_IF;

	2 : IF TUE
	     	THEN dayOk := TRUE;
		ELSE dayOk := FALSE;
	     END_IF;

      3 : IF WED
	     	THEN dayOk := TRUE;
		ELSE dayOk := FALSE;
	     END_IF;

      4 : IF THU
	     	THEN dayOk := TRUE;
		ELSE dayOk := FALSE;
	     END_IF;

      5 : IF FRI
	     	THEN dayOk := TRUE;
		ELSE dayOk := FALSE;
	     END_IF;

      6 : IF SAT
	     	THEN dayOk := TRUE;
		ELSE dayOk := FALSE;
	     END_IF;

      0 : IF SUN
	     	THEN dayOk := TRUE;
		ELSE dayOk := FALSE;
	     END_IF;

END_CASE;

(* авто *)
IF dist_manka = FALSE THEN

	(* насос *)
	IF ( ( cir2mustRun ) OR ( cir3mustRun ) OR ( cir4mustRun ) ) AND ( dayOk )
		THEN auto_pump_start := TRUE;
		ELSE auto_pump_start := FALSE;
	END_IF;

	(* клапана *)
	IF ( cir1mustRun ) AND ( dayOk )
		THEN auto_v1_open := TRUE;
		ELSE auto_v1_open := FALSE;
	END_IF;

	IF ( cir2mustRun ) AND ( dayOk )
		THEN auto_v2_open := TRUE;
		ELSE auto_v2_open := FALSE;
	END_IF;

	IF ( cir3mustRun ) AND ( dayOk )
		THEN auto_v3_open := TRUE;
		ELSE auto_v3_open := FALSE;
	END_IF;

	IF ( cir4mustRun ) AND ( dayOk )
		THEN auto_v4_open := TRUE;
		ELSE auto_v4_open := FALSE;
	END_IF;

END_IF;

(* ручное дистанционно *)
IF dist_manka  THEN

	IF ( dist_valve2 ) OR ( dist_valve3 ) OR ( dist_valve4 )
		THEN dist_pump_start := TRUE;
		ELSE dist_pump_start := FALSE;
	END_IF;

	IF dist_valve1
		THEN dist_v1_open := TRUE;
		ELSE dist_v1_open := FALSE;
	END_IF;

	IF dist_valve2
		THEN dist_v2_open := TRUE;
		ELSE dist_v2_open := FALSE;
	END_IF;

	IF dist_valve3
		THEN dist_v3_open := TRUE;
		ELSE dist_v3_open := FALSE;
	END_IF;

	IF dist_valve4
		THEN dist_v4_open := TRUE;
		ELSE dist_v4_open := FALSE;
	END_IF;

END_IF;

(* примечание: помимо дистанционного управления есть управление с галетников,
				   имеющее наивысший приоритет.
 				   управление с галетников описано в Outs 								*)
END_ACTION
ACTION Tele:
pad_PoliwTELE.0 := DI_pumpState;
pad_PoliwTELE.1 := DO_valve1;
pad_PoliwTELE.2 := DO_valve2;
pad_PoliwTELE.3 := DO_valve3;
pad_PoliwTELE.4 := DO_valve4;
pad_PoliwTELE.5 := DO_exMech;
pad_PoliwTELE.6 := DI_rainSens;
(*pad_PoliwTELE.7 := DI_humSens;*)

tele_year := TimeAndDate.Year;
tele_month := TimeAndDate.Month;
tele_day := TimeAndDate.Day;
tele_hour := TimeAndDate.Hour;
tele_minute := TimeAndDate.Minute;
END_ACTION
ACTION Times:
TimeAndDate.Day :=0;
TimeAndDate.DayOfWeek :=0;
TimeAndDate.dwHighMsec :=0;
TimeAndDate.dwLowMSecs :=0;
TimeAndDate.Milliseconds :=0;
TimeAndDate.Minute :=0;
TimeAndDate.Second :=0;
TimeAndDate.Hour :=0;
TimeAndDate.Year :=0;
TimeAndDate.Month :=0;
Sys_time.ulHigh :=0;
Sys_time.ulLow :=0;
GetTime (SystemTime:=Sys_Time , TimeDate:= TimeAndDate);


IF set_time THEN

	TimeAndDate.Minute:=setMinute;
	TimeAndDate.Second:=0;
	TimeAndDate.Hour:=setHour;
	TimeAndDate.Day:=setDay;
	TimeAndDate.Month:=setMonth;
	TimeAndDate.Year:=setYear;
	GetTime (SystemTime:=Sys_Time , TimeDate:= TimeAndDate);

END_IF;
END_ACTION
ACTION WithdrawRetain:
(*
pad_PoliwDIST := SAVE_BITS;

cir1On := save_cir1On;
cir1Off := save_cir1Off;

cir2On := save_cir2On;
cir2Off := save_cir2Off;

cir3On := save_cir3On;
cir3Off := save_cir3Off;
*)
save_cir3Off := 0;
END_ACTION

(* POU FOUNTAIN, ST *)
PROGRAM FOUNTAIN
VAR
	NO_FIRST_PASS : BOOL;
	PUNCH : WORD;

	tele_byte : BYTE;

	dist_founOn, dist_dynamic : BOOL;

	M1: BOOL;
	founT1: TON;
	M2: BOOL;
	founT2: TON;
	M3: BOOL;
	founT3: TON;
	M4: BOOL;
	founT4: TON;
	M5: BOOL;
	founT5: TON;
	M6: BOOL;
	founT6: TON;
	M7: BOOL;
	founT7: TON;
	M8: BOOL;
	founT8: TON;
	M9: BOOL;
	founT9: TON;
	M10: BOOL;
	founT10: TON;

	nodyn: BOOL;

	FPFON: R_TRIG;

	galetMode: BOOL;

(* ex-ratain*)
	staticFValue : REAL;

	founV1F: REAL;
	founV2F: REAL;
	founV3F: REAL;
	founV4F: REAL;
	founV5F: REAL;
	founV6F: REAL;
	founV7F: REAL;
	founV8F: REAL;
	founV9F: REAL;
	founV10F: REAL;

	founS1T: TIME;
	founS2T: TIME;
	founS3T: TIME;
	founS4T: TIME;
	founS5T: TIME;
	founS6T: TIME;
	founS7T: TIME;
	founS8T: TIME;
	founS9T: TIME;
	founS10T: TIME;
END_VAR

VAR RETAIN
	save_DIST : WORD;
	save_staticFValue : WORD;
	save_p1, save_p2, save_p3, save_p4, save_p5,
	save_p6, save_p7, save_p8, save_p9, save_p10 : WORD;

END_VAR
VAR (* helpers for the ST form of the networks *)
	_p1 : BOOL;
	_p2 : BOOL;
	_p3 : BOOL;
	_p4 : BOOL;
	_p5 : BOOL;
	_p6 : BOOL;
	_p7 : BOOL;
	_p8 : BOOL;
	_p9 : BOOL;
	_p10 : BOOL;
END_VAR
(* 				first pass 				*)
IF NO_FIRST_PASS = FALSE
	THEN WithdrawRetain;
	PUNCH := 1023;
	Obtaining;
	PUNCH := 0;
	NO_FIRST_PASS := TRUE;
END_IF;

(*			    main cycle		  		*)
PUNCH := 0;

CheckNewVal;

IF PUNCH > 0
	THEN Obtaining;
END_IF;


IF dist_dynamic
	THEN nodyn := FALSE;
	ELSE nodyn := TRUE;
END_IF;

IF ( founV1F = 0.0 ) AND
	( founV2F = 0.0 ) AND
	( founV3F = 0.0 ) AND
	( founV4F = 0.0 ) AND
	( founV5F = 0.0 ) AND
	( founV6F = 0.0 ) AND
	( founV7F = 0.0 ) AND
	( founV8F = 0.0 ) AND
	( founV9F = 0.0 ) AND
	( founV10F = 0.0 )
THEN
	nodyn := TRUE;
END_IF;

IF DI_staticMode
	THEN nodyn := TRUE;
END_IF;

IF DI_dynamicMode
	THEN nodyn := FALSE;
END_IF;

AOvalues;

PumpCtrl;

Forwarding;
END_PROGRAM
ACTION AOvalues:
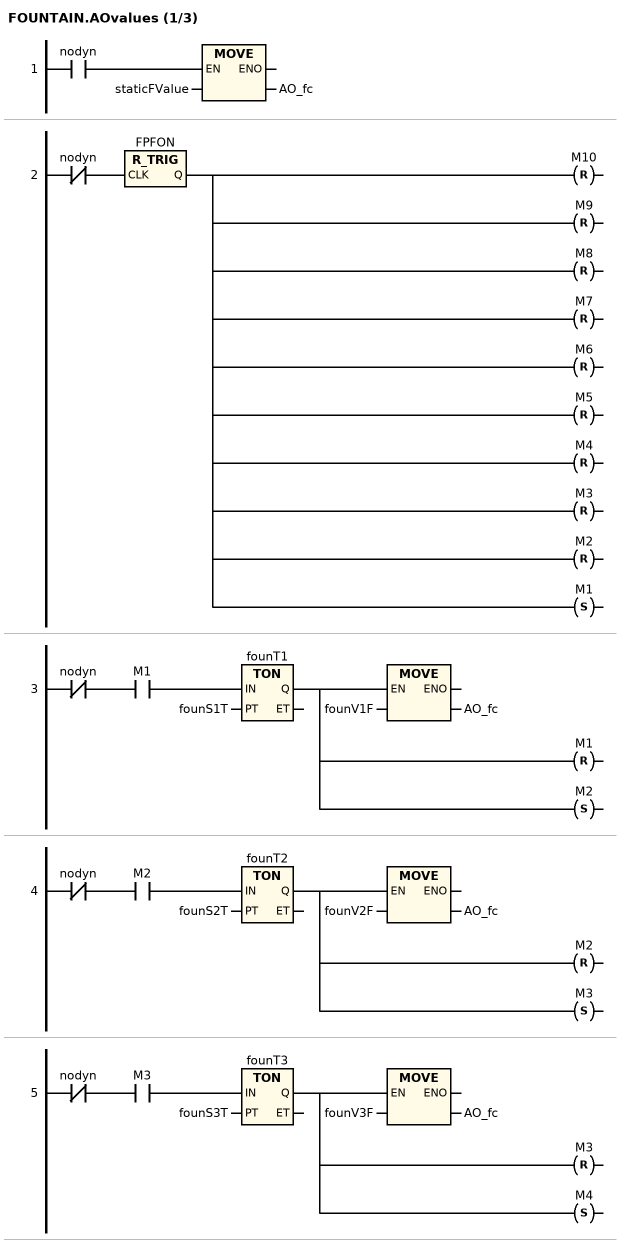
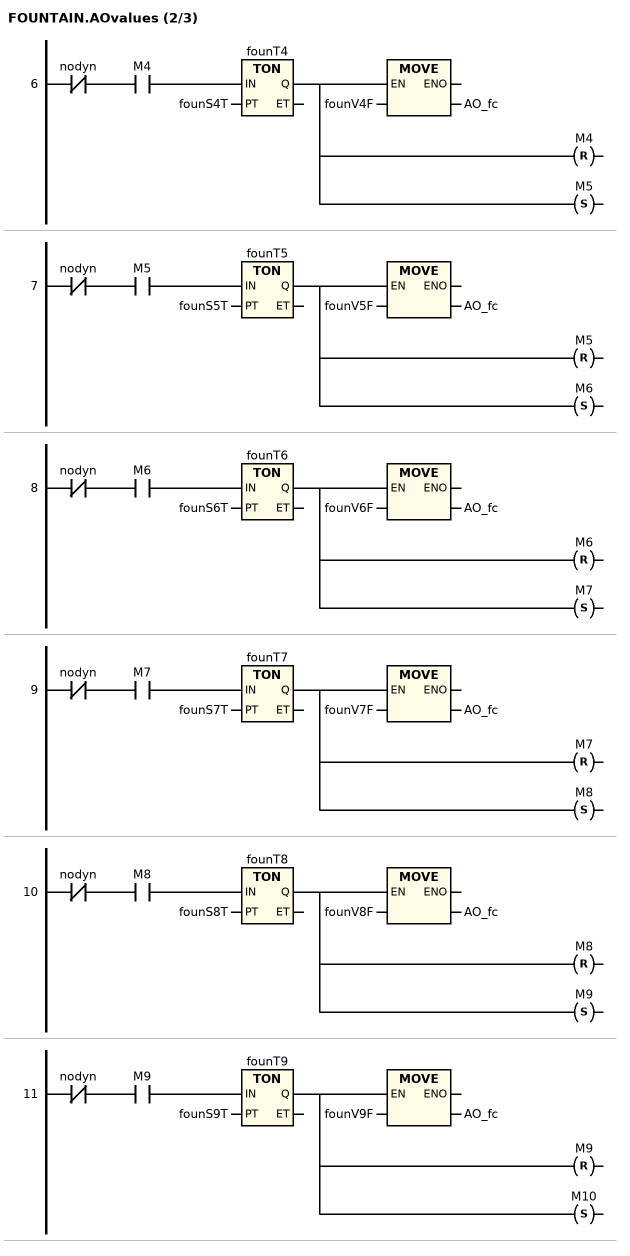
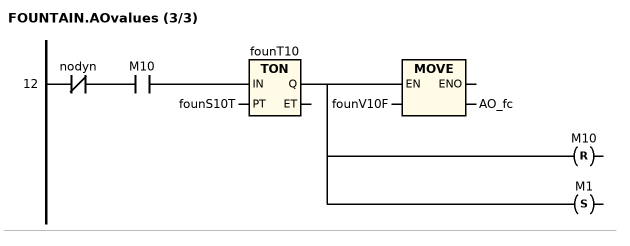
_LD_ (* Ladder Diagram *)
NETWORK 1
	[nodyn]
		EN --- MOVE(staticFValue) => AO_fc
NETWORK 2
	[/nodyn] - FPFON:R_TRIG(CLK: *) --- (R M10) (R M9) (R M8) (R M7) (R M6) (R M5) (R M4) (R M3) (R M2) (S M1)
NETWORK 3
	[/nodyn] - [M1] - founT1:TON(IN: *, PT: founS1T) --- (R M1) (S M2)
		EN --- MOVE(founV1F) => AO_fc
NETWORK 4
	[/nodyn] - [M2] - founT2:TON(IN: *, PT: founS2T) --- (R M2) (S M3)
		EN --- MOVE(founV2F) => AO_fc
NETWORK 5
	[/nodyn] - [M3] - founT3:TON(IN: *, PT: founS3T) --- (R M3) (S M4)
		EN --- MOVE(founV3F) => AO_fc
NETWORK 6
	[/nodyn] - [M4] - founT4:TON(IN: *, PT: founS4T) --- (R M4) (S M5)
		EN --- MOVE(founV4F) => AO_fc
NETWORK 7
	[/nodyn] - [M5] - founT5:TON(IN: *, PT: founS5T) --- (R M5) (S M6)
		EN --- MOVE(founV5F) => AO_fc
NETWORK 8
	[/nodyn] - [M6] - founT6:TON(IN: *, PT: founS6T) --- (R M6) (S M7)
		EN --- MOVE(founV6F) => AO_fc
NETWORK 9
	[/nodyn] - [M7] - founT7:TON(IN: *, PT: founS7T) --- (R M7) (S M8)
		EN --- MOVE(founV7F) => AO_fc
NETWORK 10
	[/nodyn] - [M8] - founT8:TON(IN: *, PT: founS8T) --- (R M8) (S M9)
		EN --- MOVE(founV8F) => AO_fc
NETWORK 11
	[/nodyn] - [M9] - founT9:TON(IN: *, PT: founS9T) --- (R M9) (S M10)
		EN --- MOVE(founV9F) => AO_fc
NETWORK 12
	[/nodyn] - [M10] - founT10:TON(IN: *, PT: founS10T) --- (R M10) (S M1)
		EN --- MOVE(founV10F) => AO_fc
_END_LD_
(* the same logic as Structured Text *)
(* Network 1 *)
IF nodyn THEN
	AO_fc := staticFValue;
END_IF;
(* Network 2 *)
FPFON(CLK := NOT nodyn);
IF FPFON.Q THEN M10 := FALSE; M9 := FALSE; M8 := FALSE; M7 := FALSE; M6 := FALSE; M5 := FALSE; M4 := FALSE; M3 := FALSE; M2 := FALSE; M1 := TRUE; END_IF;
(* Network 3 *)
founT1(IN := NOT nodyn AND M1, PT := founS1T);
_p1 := founT1.Q;
IF _p1 THEN
	AO_fc := founV1F;
END_IF;
IF _p1 THEN M1 := FALSE; M2 := TRUE; END_IF;
(* Network 4 *)
founT2(IN := NOT nodyn AND M2, PT := founS2T);
_p2 := founT2.Q;
IF _p2 THEN
	AO_fc := founV2F;
END_IF;
IF _p2 THEN M2 := FALSE; M3 := TRUE; END_IF;
(* Network 5 *)
founT3(IN := NOT nodyn AND M3, PT := founS3T);
_p3 := founT3.Q;
IF _p3 THEN
	AO_fc := founV3F;
END_IF;
IF _p3 THEN M3 := FALSE; M4 := TRUE; END_IF;
(* Network 6 *)
founT4(IN := NOT nodyn AND M4, PT := founS4T);
_p4 := founT4.Q;
IF _p4 THEN
	AO_fc := founV4F;
END_IF;
IF _p4 THEN M4 := FALSE; M5 := TRUE; END_IF;
(* Network 7 *)
founT5(IN := NOT nodyn AND M5, PT := founS5T);
_p5 := founT5.Q;
IF _p5 THEN
	AO_fc := founV5F;
END_IF;
IF _p5 THEN M5 := FALSE; M6 := TRUE; END_IF;
(* Network 8 *)
founT6(IN := NOT nodyn AND M6, PT := founS6T);
_p6 := founT6.Q;
IF _p6 THEN
	AO_fc := founV6F;
END_IF;
IF _p6 THEN M6 := FALSE; M7 := TRUE; END_IF;
(* Network 9 *)
founT7(IN := NOT nodyn AND M7, PT := founS7T);
_p7 := founT7.Q;
IF _p7 THEN
	AO_fc := founV7F;
END_IF;
IF _p7 THEN M7 := FALSE; M8 := TRUE; END_IF;
(* Network 10 *)
founT8(IN := NOT nodyn AND M8, PT := founS8T);
_p8 := founT8.Q;
IF _p8 THEN
	AO_fc := founV8F;
END_IF;
IF _p8 THEN M8 := FALSE; M9 := TRUE; END_IF;
(* Network 11 *)
founT9(IN := NOT nodyn AND M9, PT := founS9T);
_p9 := founT9.Q;
IF _p9 THEN
	AO_fc := founV9F;
END_IF;
IF _p9 THEN M9 := FALSE; M10 := TRUE; END_IF;
(* Network 12 *)
founT10(IN := NOT nodyn AND M10, PT := founS10T);
_p10 := founT10.Q;
IF _p10 THEN
	AO_fc := founV10F;
END_IF;
IF _p10 THEN M10 := FALSE; M1 := TRUE; END_IF;
END_ACTION
ACTION CheckNewVal:
IF save_DIST <> FounDIST
	THEN save_DIST:= FounDIST;
			PUNCH.0 := TRUE;
END_IF;

IF save_p1 <> p1
	THEN save_p1 := p1;
			PUNCH.1 := TRUE;
END_IF;

IF save_p2 <> p2
	THEN save_p2 := p2;
			PUNCH.2 := TRUE;
END_IF;

IF save_p3 <> p3
	THEN save_p3 := p3;
			PUNCH.3 := TRUE;
END_IF;

IF save_p4 <> p4
	THEN save_p4 := p4;
			PUNCH.4 := TRUE;
END_IF;

IF save_p5 <> p5
	THEN save_p5 := p5;
			PUNCH.5 := TRUE;
END_IF;

IF save_p6 <> p6
	THEN save_p6 := p6;
			PUNCH.6 := TRUE;
END_IF;

IF save_p7 <> p7
	THEN save_p7 := p7;
			PUNCH.7 := TRUE;
END_IF;

IF save_p8 <> p8
	THEN save_p8 := p8;
			PUNCH.8 := TRUE;
END_IF;

IF save_p9 <> p9
	THEN save_p9 := p9;
			PUNCH.9 := TRUE;
END_IF;

IF save_p10 <> p10
	THEN save_p10 := p10;
			PUNCH.10 := TRUE;
END_IF;

IF save_staticFValue <> dist_staticFValue
	THEN save_staticFValue := dist_staticFvalue;
			PUNCH.11 := TRUE;
END_IF;
END_ACTION
ACTION Forwarding:
(*
tele_byte.0 := DO_pump;
tele_byte.1 := DI_staticMode;
tele_byte.2 := DI_dynamicMode;
*)
FounTELE := REAL_TO_WORD ( AO_fc * 10 );
END_ACTION
ACTION Obtaining:
IF PUNCH.0 THEN
	dist_founOn := save_DIST.0;
	dist_dynamic := save_DIST.1;
(*
	staticFValue := BYTE_TO_REAL (
							WORD_TO_BYTE ( save_DIST / 256 ) ) / 10;
*)
	PUNCH.0 := FALSE;
END_IF;

IF PUNCH.11 THEN
	staticFValue := WORD_TO_REAL ( save_staticFValue ) / 10;
	PUNCH.11 := FALSE;
END_IF;

(*
	lo,hi : byte
	w : word

	lo := word_to_byte(w)
	hi := word_to_byte(w/256)
	w := 256*hi + lo 
*)

IF PUNCH.1 THEN
	founV1F := BYTE_TO_REAL ( WORD_TO_BYTE ( save_p1 ) ) / 10;
	founS1T := WORD_TO_TIME ( WORD_TO_BYTE ( save_p1 / 256 ) * 1000 );
	PUNCH.1 := FALSE;
END_IF;

IF PUNCH.2 THEN
	founV2F := BYTE_TO_REAL ( WORD_TO_BYTE ( save_p2 ) ) / 10;
	founS2T := WORD_TO_TIME ( WORD_TO_BYTE ( save_p2 / 256 ) * 1000 );
	PUNCH.2 := FALSE;
END_IF;

IF PUNCH.3 THEN
	founV3F := BYTE_TO_REAL ( WORD_TO_BYTE ( save_p3 ) ) /10;
	founS3T := WORD_TO_TIME ( WORD_TO_BYTE ( save_p3 / 256 ) * 1000 );
	PUNCH.3 := FALSE;
END_IF;

IF PUNCH.4 THEN
	founV4F := BYTE_TO_REAL ( WORD_TO_BYTE ( save_p4 ) ) /10;
	founS4T := WORD_TO_TIME ( WORD_TO_BYTE ( save_p4 / 256 ) * 1000 );
	PUNCH.4 := FALSE;
END_IF;

IF PUNCH.5 THEN
	founV5F := BYTE_TO_REAL ( WORD_TO_BYTE ( save_p5 ) ) /10;
	founS5T := WORD_TO_TIME ( WORD_TO_BYTE ( save_p5 / 256 ) * 1000 );
	PUNCH.5 := FALSE;
END_IF;

IF PUNCH.6 THEN
	founV6F := BYTE_TO_REAL ( WORD_TO_BYTE ( save_p6 ) ) /10;
	founS6T := WORD_TO_TIME ( WORD_TO_BYTE ( save_p6 / 256 ) * 1000 );
	PUNCH.6 := FALSE;
END_IF;

IF PUNCH.7 THEN
	founV7F := BYTE_TO_REAL ( WORD_TO_BYTE ( save_p7 ) ) /10;
	founS7T := WORD_TO_TIME ( WORD_TO_BYTE ( save_p7 / 256 ) * 1000 );
	PUNCH.7 := FALSE;
END_IF;

IF PUNCH.8 THEN
	founV8F := BYTE_TO_REAL ( WORD_TO_BYTE ( save_p8 ) ) /10;
	founS8T := WORD_TO_TIME ( WORD_TO_BYTE ( save_p8 / 256 ) * 1000 );
	PUNCH.8 := FALSE;
END_IF;

IF PUNCH.9 THEN
	founV9F := BYTE_TO_REAL ( WORD_TO_BYTE ( save_p9 ) ) /10;
	founS9T := WORD_TO_TIME ( WORD_TO_BYTE ( save_p9 / 256 ) * 1000 );
	PUNCH.9 := FALSE;
END_IF;

IF PUNCH.10 THEN
	founV10F := BYTE_TO_REAL ( WORD_TO_BYTE ( save_p10 ) ) /10;
	founS10T := WORD_TO_TIME ( WORD_TO_BYTE ( save_p10 / 256 ) * 1000 );
	PUNCH.10 := FALSE;
END_IF;
END_ACTION
ACTION PumpCtrl:
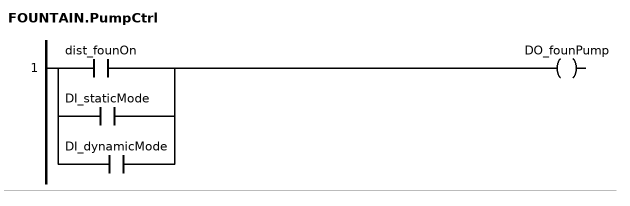
_LD_ (* Ladder Diagram *)
NETWORK 1
	{ [dist_founOn] | [DI_staticMode] | [DI_dynamicMode] } --- (DO_founPump)
_END_LD_
(* the same logic as Structured Text *)
(* Network 1 *)
DO_founPump := dist_founOn OR DI_staticMode OR DI_dynamicMode;
END_ACTION
ACTION WithdrawRetain:
(*
FounDIST := save_DIST;

p1 := save_p1;
p2 := save_p2;
p3 := save_p3;
p4 := save_p4;
p5 := save_p5;
p6 := save_p6;
p7 := save_p7;
p8 := save_p8;
p9 := save_p9;
p10 := save_p10;
*)

save_p10 := 0;
END_ACTION

(* POU TRM, ST *)
PROGRAM TRM
VAR
	PUNCH : WORD;
	NO_FIRST_PASS : BOOL;

	trm1_ch1_dayHH, trm1_ch1_dayMM, trm1_ch1_nightHH, trm1_ch1_nightMM,
	trm1_ch2_dayHH, trm1_ch2_dayMM, trm1_ch2_nightHH, trm1_ch2_nightMM,
	trm2_ch1_dayHH, trm2_ch1_dayMM, trm2_ch1_nightHH, trm2_ch1_nightMM,
	trm2_ch2_dayHH, trm2_ch2_dayMM, trm2_ch2_nightHH, trm2_ch2_nightMM : BYTE;
END_VAR

VAR RETAIN
	trm1_set1_save, trm1_set2_save : WORD;
	trm2_set1_save, trm2_set2_save : WORD;

	trm1_set1_saev, trm1_set2_saev : WORD;
	trm2_set1_saev, trm2_set2_saev : WORD;

	trm1_ch1_day_save, trm1_ch1_night_save,
	trm1_ch2_day_save, trm1_ch2_night_save,
	trm2_ch1_day_save, trm2_ch1_night_save,
	trm2_ch2_day_save, trm2_ch2_night_save : WORD;

	trm1_ch1_dayVal_save, trm1_ch1_dayNight_save: WORD;
	trm1_ch2_dayVal_save, trm1_ch2_dayNight_save: WORD;
	trm2_ch1_dayVal_save, trm2_ch1_dayNight_save: WORD;
	trm2_ch2_dayVal_save, trm2_ch2_dayNight_save: WORD;

	trm1_ch1_nightVal_save, trm1_ch1_nightNight_save: WORD;
	trm1_ch2_nightVal_save, trm1_ch2_nightNight_save: WORD;
	trm2_ch1_nightVal_save, trm2_ch1_nightNight_save: WORD;
	trm2_ch2_nightVal_save, trm2_ch2_nightNight_save: WORD;
END_VAR
IF NO_FIRST_PASS = FALSE
	THEN WithdrawRetain;
	NO_FIRST_PASS := TRUE;
END_IF;

PUNCH := 0;

CheckNewVal;

IF PUNCH > 0 THEN
	Refresh;
END_IF;

UnpackTime;

Schedule;

Transfer;
END_PROGRAM
ACTION CheckNewVal:
(*				TRM 1				*)
IF trm1_set1_save <> pad_trm1_set1
	THEN trm1_set1_save := pad_trm1_set1;
	PUNCH.0 := TRUE;
END_IF;

IF trm1_set2_save <> pad_trm1_set2
	THEN trm1_set2_save := pad_trm1_set2;
	PUNCH.1 := TRUE;
END_IF;



IF trm1_set1_saev <> trm1_set1_read
	THEN trm1_set1_saev := trm1_set1_read;
	PUNCH.2 := TRUE;
END_IF;

IF trm1_set2_saev <> trm1_set2_read
	THEN trm1_set2_saev := trm1_set2_read;
	PUNCH.3 := TRUE;
END_IF;



(*				TRM 2				*)
IF trm2_set1_save <> pad_trm2_set1
	THEN trm2_set1_save := pad_trm2_set1;
	PUNCH.4 := TRUE;
END_IF;

IF trm2_set2_save <> pad_trm2_set2
	THEN trm2_set2_save := pad_trm2_set2;
	PUNCH.5 := TRUE;
END_IF;



IF trm2_set1_saev <> trm2_set1_read
	THEN trm2_set1_saev := trm2_set1_read;
	PUNCH.6 := TRUE;
END_IF;

IF trm2_set2_saev <> trm2_set2_read
	THEN trm2_set2_saev := trm2_set2_read;
	PUNCH.7 := TRUE;
END_IF;


(* all day~ *)
IF trm1_ch1_day_save <> trm1_ch1_day
	THEN trm1_ch1_day_save := trm1_ch1_day;
END_IF;

IF trm1_ch2_day_save <> trm1_ch2_day
	THEN trm1_ch2_day_save := trm1_ch2_day;
END_IF;

IF trm2_ch1_day_save <> trm2_ch1_day
	THEN trm2_ch1_day_save := trm2_ch1_day;
END_IF;

IF trm2_ch2_day_save <> trm2_ch2_day
	THEN trm2_ch2_day_save := trm2_ch2_day;
END_IF;


(* all night~ *)
IF trm1_ch1_night_save <> trm1_ch1_night
	THEN trm1_ch1_night_save := trm1_ch1_night;
END_IF;

IF trm1_ch2_night_save <> trm1_ch2_night
	THEN trm1_ch2_night_save := trm1_ch2_night;
END_IF;

IF trm2_ch1_night_save <> trm2_ch1_night
	THEN trm2_ch1_night_save := trm2_ch1_night;
END_IF;

IF trm2_ch2_night_save <> trm2_ch2_night
	THEN trm2_ch2_night_save := trm2_ch2_night;
END_IF;

(* all day~ *)
IF trm1_ch1_dayVal_save <> trm1_ch1_dayVal
	THEN trm1_ch1_dayVal_save := trm1_ch1_dayVal;
END_IF;

IF trm1_ch2_dayVal_save <> trm1_ch2_dayVal
	THEN trm1_ch2_dayVal_save := trm1_ch2_dayVal;
END_IF;

IF trm2_ch1_dayVal_save <> trm2_ch1_dayVal
	THEN trm2_ch1_dayVal_save := trm2_ch1_dayVal;
END_IF;

IF trm2_ch2_dayVal_save <> trm2_ch2_dayVal
	THEN trm2_ch2_dayVal_save := trm2_ch2_dayVal;
END_IF;

(* all night~ *)
IF trm1_ch1_nightVal_save <> trm1_ch1_nightVal
	THEN trm1_ch1_nightVal_save := trm1_ch1_nightVal;
END_IF;

IF trm1_ch2_nightVal_save <> trm1_ch2_nightVal
	THEN trm1_ch2_nightVal_save := trm1_ch2_nightVal;
END_IF;

IF trm2_ch1_nightVal_save <> trm2_ch1_nightVal
	THEN trm2_ch1_nightVal_save := trm2_ch1_nightVal;
END_IF;

IF trm2_ch2_nightVal_save <> trm2_ch2_nightVal
	THEN trm2_ch2_nightVal_save := trm2_ch2_nightVal;
END_IF;
END_ACTION
ACTION Refresh:
(*			ТРМ 1			*)
IF PUNCH.0
	THEN trm1_set1_write := trm1_set1_save;
	trm1_set1_saev := trm1_set1_save;
	PUNCH.0 := FALSE;
END_IF;

IF PUNCH.1
	THEN trm1_set2_write := trm1_set2_save;
	trm1_set2_saev := trm1_set2_save;
 	PUNCH.1 := FALSE;
END_IF;


IF PUNCH.2
	THEN pad_trm1_set1 := trm1_set1_saev;
	trm1_set1_save := trm1_set1_saev;
	PUNCH.2 := FALSE;
END_IF;

IF PUNCH.3
	THEN pad_trm1_set2 := trm1_set2_saev;
	trm1_set2_save := trm1_set2_saev;
	PUNCH.3 := FALSE;
END_IF;


(*				ТРМ 2 				*)
IF PUNCH.4
	THEN trm2_set1_write := trm2_set1_save;
	trm2_set1_saev := trm2_set1_save;
	PUNCH.4 := FALSE;
END_IF;

IF PUNCH.5
	THEN trm2_set2_write := trm2_set2_save;
	trm2_set2_saev := trm2_set2_save;
	PUNCH.5 := FALSE;
END_IF;


IF PUNCH.6
	THEN pad_trm2_set1 := trm2_set1_saev;
	trm2_set1_save := trm2_set1_saev;
	PUNCH.6 := FALSE;
END_IF;

IF PUNCH.7
	THEN pad_trm2_set2 := trm2_set2_saev;
	trm2_set2_save := trm2_set2_saev;
	PUNCH.7 := FALSE;
END_IF;
END_ACTION
ACTION Schedule:
(* all day~ *)
IF ( trm1_ch1_dayHH = TimeAndDate.Hour ) AND ( trm1_ch1_dayMM = TimeAndDate.Minute ) AND ( TimeAndDate.Second = 0 )
	THEN pad_trm1_set1 := trm1_ch1_dayVal;
END_IF;

IF ( trm1_ch2_dayHH = TimeAndDate.Hour ) AND ( trm1_ch2_dayMM = TimeAndDate.Minute ) AND ( TimeAndDate.Second = 0 )
	THEN pad_trm1_set2 := trm1_ch2_dayVal;
END_IF;

IF ( trm2_ch1_dayHH = TimeAndDate.Hour ) AND ( trm2_ch1_dayMM = TimeAndDate.Minute ) AND ( TimeAndDate.Second = 0 )
	THEN pad_trm2_set1 := trm2_ch1_dayVal;
END_IF;

IF ( trm2_ch2_dayHH = TimeAndDate.Hour ) AND ( trm2_ch2_dayMM = TimeAndDate.Minute ) AND ( TimeAndDate.Second = 0 )
	THEN pad_trm2_set2 := trm2_ch2_dayVal;
END_IF;

(* all night~ *)
IF ( trm1_ch1_nightHH = TimeAndDate.Hour ) AND ( trm1_ch1_nightMM = TimeAndDate.Minute ) AND ( TimeAndDate.Second = 0 )
	THEN pad_trm1_set1 := trm1_ch1_nightVal;
END_IF;

IF ( trm1_ch2_nightHH = TimeAndDate.Hour ) AND ( trm1_ch2_nightMM = TimeAndDate.Minute ) AND ( TimeAndDate.Second = 0 )
	THEN pad_trm1_set2 := trm1_ch2_nightVal;
END_IF;

IF ( trm2_ch1_nightHH = TimeAndDate.Hour ) AND ( trm2_ch1_nightMM = TimeAndDate.Minute ) AND ( TimeAndDate.Second = 0 )
	THEN pad_trm2_set1 := trm2_ch1_nightVal;
END_IF;

IF ( trm2_ch2_nightHH = TimeAndDate.Hour ) AND ( trm2_ch2_nightMM = TimeAndDate.Minute ) AND ( TimeAndDate.Second = 0 )
	THEN pad_trm2_set2 := trm2_ch2_nightVal;
END_IF;
END_ACTION
ACTION Transfer:
pad_trm1_ch1 := trm1_ch1;
pad_trm1_ch2 := trm1_ch2;

pad_trm2_ch1 := trm2_ch1;
pad_trm2_ch2 := trm2_ch2;

IF (trm1_out1 = 1000)
	THEN TRMOUTS.0 := TRUE;
	ELSE TRMOUTS.0 := FALSE;
END_IF;

IF (trm1_out2 = 1000)
	THEN TRMOUTS.1 := TRUE;
	ELSE TRMOUTS.1 := FALSE;
END_IF;

IF (trm2_out1 = 1000)
	THEN TRMOUTS.2 := TRUE;
	ELSE TRMOUTS.2 := FALSE;
END_IF;

IF (trm2_out2 = 1000)
	THEN TRMOUTS.3:= TRUE;
	ELSE TRMOUTS.3:= FALSE;
END_IF;
END_ACTION
ACTION UnpackTime:
(*
	lo,hi : byte
	w : word

	lo := word_to_byte(w)
	hi := word_to_byte(w/256)
	w := 256*hi + lo 
*)

trm1_ch1_dayHH := WORD_TO_BYTE ( trm1_ch1_day_save );
trm1_ch1_dayMM := WORD_TO_BYTE ( trm1_ch1_day_save / 256 );

trm1_ch2_dayHH := WORD_TO_BYTE ( trm1_ch2_day_save );
trm1_ch2_dayMM := WORD_TO_BYTE ( trm1_ch2_day_save / 256 );

trm2_ch1_dayHH := WORD_TO_BYTE ( trm2_ch1_day_save );
trm2_ch1_dayMM := WORD_TO_BYTE ( trm2_ch1_day_save / 256 );

trm2_ch2_dayHH := WORD_TO_BYTE ( trm2_ch2_day_save );
trm2_ch2_dayMM := WORD_TO_BYTE ( trm2_ch2_day_save / 256 );


trm1_ch1_nightHH := WORD_TO_BYTE ( trm1_ch1_night_save );
trm1_ch1_nightMM := WORD_TO_BYTE ( trm1_ch1_night_save / 256 );

trm1_ch2_nightHH := WORD_TO_BYTE ( trm1_ch2_night_save );
trm1_ch2_nightMM := WORD_TO_BYTE ( trm1_ch2_night_save / 256 );

trm2_ch1_nightHH := WORD_TO_BYTE ( trm2_ch1_night_save );
trm2_ch1_nightMM := WORD_TO_BYTE ( trm2_ch1_night_save / 256 );

trm2_ch2_nightHH := WORD_TO_BYTE ( trm2_ch2_night_save );
trm2_ch2_nightMM := WORD_TO_BYTE ( trm2_ch2_night_save / 256 );
END_ACTION
ACTION WithdrawRetain:
(*
pad_trm1_set1 := trm1_set1_save;
pad_trm1_set2 := trm1_set2_save;


pad_trm2_set1 := trm2_set1_save;
pad_trm2_set2 := trm2_set2_save;

trm1_ch1_day := trm1_ch1_day_save;
trm1_ch1_night := trm1_ch1_night_save;

trm1_ch2_day := trm1_ch2_day_save;
trm1_ch2_night := trm1_ch2_night_save;

trm2_ch1_day := trm2_ch1_day_save;
trm2_ch1_night := trm2_ch1_night_save;

trm2_ch2_day := trm2_ch2_day_save;
trm2_ch2_night := trm2_ch2_night_save;

trm1_ch1_dayVal := trm1_ch1_dayVal_save;
trm1_ch2_dayVal := trm1_ch2_dayVal_save;

trm2_ch1_dayVal := trm2_ch1_dayVal_save;
trm2_ch2_dayVal := trm2_ch2_dayVal_save;


trm1_ch1_nightVal := trm1_ch1_nightVal_save;
trm1_ch2_nightVal := trm1_ch2_nightVal_save;

trm2_ch1_nightVal := trm2_ch1_nightVal_save;
trm2_ch2_nightVal := trm2_ch2_nightVal_save;
(*
trm1_ch1_night := trm1_ch1_night_save;
trm1_ch2_night := trm1_ch2_night_save;
trm2_ch1_night := trm2_ch1_night_save;
trm2_ch2_night := trm2_ch2_night_save;


trm1_ch1_day := trm1_ch1_day_save;
trm1_ch2_day := trm1_ch2_day_save;
trm2_ch1_day := trm2_ch1_day_save;
trm2_ch2_day := trm2_ch2_day_save;
*)
*)
trm2_ch2_day_save := 0;
END_ACTION

(* POU LIGHT, ST *)
PROGRAM LIGHT
VAR
	NO_FIRST_PASS : BOOL;

	boolLamp1: BOOL;
	boolLamp2: BOOL;
	boolLamp3: BOOL;
	FP1: R_TRIG;
	FP2: R_TRIG;
	FP3: R_TRIG;
	FN1: F_TRIG;
	FP4: R_TRIG;
	FP5: R_TRIG;
	FP6: R_TRIG;
	FN2: F_TRIG;
	FP7: R_TRIG;
	FP8: R_TRIG;
	FP9: R_TRIG;
	FN3: F_TRIG;

	lamp1OnHH, lamp1OnMM, lamp1OffHH, lamp1OffMM,
	lamp2OnHH, lamp2OnMM, lamp2OffHH, lamp2OffMM,
	lamp3OnHH, lamp3OnMM, lamp3OffHH, lamp3OffMM : BYTE;
END_VAR
VAR RETAIN

	diBuf1: BOOL;
	mxBuf1: BOOL;
	mx1: BOOL;
	dx1: BOOL;

	diBuf2: BOOL;
	mxBuf2: BOOL;
	mx2: BOOL;
	dx2: BOOL;


	diBuf3: BOOL;
	mxBuf3: BOOL;
	mx3: BOOL;
	dx3: BOOL;

	preDoLamp1 : BOOL;
	timeDoLamp1: BOOL;

	preDoLamp2 : BOOL;
	timeDoLamp2: BOOL;

	preDoLamp3 : BOOL;
	timeDoLamp3: BOOL;


	dim1_save, dim2_save, dim3_save : WORD;

	lamp1On_save, lamp1Off_save, lamp2On_save, lamp2Off_save,
	lamp3On_save, lamp3Off_save : WORD;


END_VAR
VAR (* helpers for the ST form of the networks *)
	_p1 : BOOL;
	_p2 : BOOL;
	_p3 : BOOL;
	_p4 : BOOL;
	_p5 : BOOL;
	_p6 : BOOL;
	_p7 : BOOL;
	_p8 : BOOL;
	_p9 : BOOL;
	_p10 : BOOL;
	_p11 : BOOL;
	_p12 : BOOL;
END_VAR
IF NO_FIRST_PASS = FALSE
	THEN WithdrawRetain;
			NO_FIRST_PASS := TRUE;
END_IF;

CheckNewValue;

AO_dim1 := WORD_TO_REAL ( dim1 ) / 10;
AO_dim2 := WORD_TO_REAL ( dim2 ) / 10;
AO_dim3 := WORD_TO_REAL ( dim3 ) / 10;

UnpackTime;
Schedule;
Lamp1;
Lamp2;
Lamp3;

DistLamp;
ForwardLampState;
END_PROGRAM
ACTION CheckNewValue:
IF dim1_save <> dim1
	THEN dim1_save := dim1;
END_IF;

IF dim2_save <> dim2
	THEN dim2_save := dim2;
END_IF;

IF dim3_save <> dim3
	THEN dim3_save := dim3;
END_IF;

IF lamp1On_save <> lamp1On
	THEN lamp1On_save := lamp1On;
END_IF;


IF lamp1Off_save <> lamp1Off
	THEN lamp1Off_save := lamp1Off;
END_IF;

IF lamp2On_save <> lamp2On
	THEN lamp2On_save := lamp2On;
END_IF;


IF lamp2Off_save <> lamp2Off
	THEN lamp2Off_save := lamp2Off;
END_IF;

IF lamp3On_save <> lamp3On
	THEN lamp3On_save := lamp3On;
END_IF;


IF lamp3Off_save <> lamp3Off
	THEN lamp3Off_save := lamp3Off;
END_IF;
END_ACTION
ACTION DistLamp:
boolLamp1 := dist_LAMP.0;
boolLamp2 := dist_LAMP.1;
boolLamp3 := dist_LAMP.2;
END_ACTION
ACTION ForwardLampState:
tele_LAMP.0 := DO_lamp1;
tele_LAMP.1 := DO_lamp2;
tele_LAMP.2 := DO_lamp3;

tele_lamp.10 := DO_founPump;
END_ACTION
ACTION Lamp1:
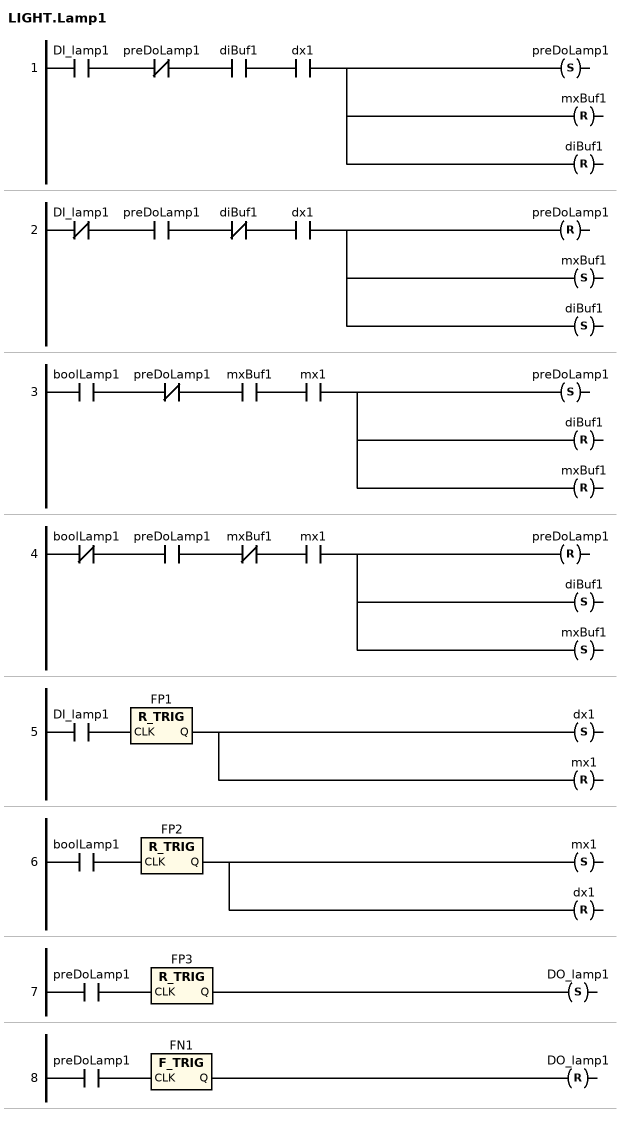
_LD_ (* Ladder Diagram *)
NETWORK 1
	[DI_lamp1] - [/preDoLamp1] - [diBuf1] - [dx1] --- (S preDoLamp1) (R mxBuf1) (R diBuf1)
NETWORK 2
	[/DI_lamp1] - [preDoLamp1] - [/diBuf1] - [dx1] --- (R preDoLamp1) (S mxBuf1) (S diBuf1)
NETWORK 3
	[boolLamp1] - [/preDoLamp1] - [mxBuf1] - [mx1] --- (S preDoLamp1) (R diBuf1) (R mxBuf1)
NETWORK 4
	[/boolLamp1] - [preDoLamp1] - [/mxBuf1] - [mx1] --- (R preDoLamp1) (S diBuf1) (S mxBuf1)
NETWORK 5
	[DI_lamp1] - FP1:R_TRIG(CLK: *) --- (S dx1) (R mx1)
NETWORK 6
	[boolLamp1] - FP2:R_TRIG(CLK: *) --- (S mx1) (R dx1)
NETWORK 7
	[preDoLamp1] - FP3:R_TRIG(CLK: *) --- (S DO_lamp1)
NETWORK 8
	[preDoLamp1] - FN1:F_TRIG(CLK: *) --- (R DO_lamp1)
_END_LD_
(* the same logic as Structured Text *)
(* Network 1 *)
_p1 := DI_lamp1 AND NOT preDoLamp1 AND diBuf1 AND dx1;
IF _p1 THEN preDoLamp1 := TRUE; mxBuf1 := FALSE; diBuf1 := FALSE; END_IF;
(* Network 2 *)
_p2 := NOT DI_lamp1 AND preDoLamp1 AND NOT diBuf1 AND dx1;
IF _p2 THEN preDoLamp1 := FALSE; mxBuf1 := TRUE; diBuf1 := TRUE; END_IF;
(* Network 3 *)
_p3 := boolLamp1 AND NOT preDoLamp1 AND mxBuf1 AND mx1;
IF _p3 THEN preDoLamp1 := TRUE; diBuf1 := FALSE; mxBuf1 := FALSE; END_IF;
(* Network 4 *)
_p4 := NOT boolLamp1 AND preDoLamp1 AND NOT mxBuf1 AND mx1;
IF _p4 THEN preDoLamp1 := FALSE; diBuf1 := TRUE; mxBuf1 := TRUE; END_IF;
(* Network 5 *)
FP1(CLK := DI_lamp1);
IF FP1.Q THEN dx1 := TRUE; mx1 := FALSE; END_IF;
(* Network 6 *)
FP2(CLK := boolLamp1);
IF FP2.Q THEN mx1 := TRUE; dx1 := FALSE; END_IF;
(* Network 7 *)
FP3(CLK := preDoLamp1);
IF FP3.Q THEN DO_lamp1 := TRUE; END_IF;
(* Network 8 *)
FN1(CLK := preDoLamp1);
IF FN1.Q THEN DO_lamp1 := FALSE; END_IF;
END_ACTION
ACTION Lamp2:
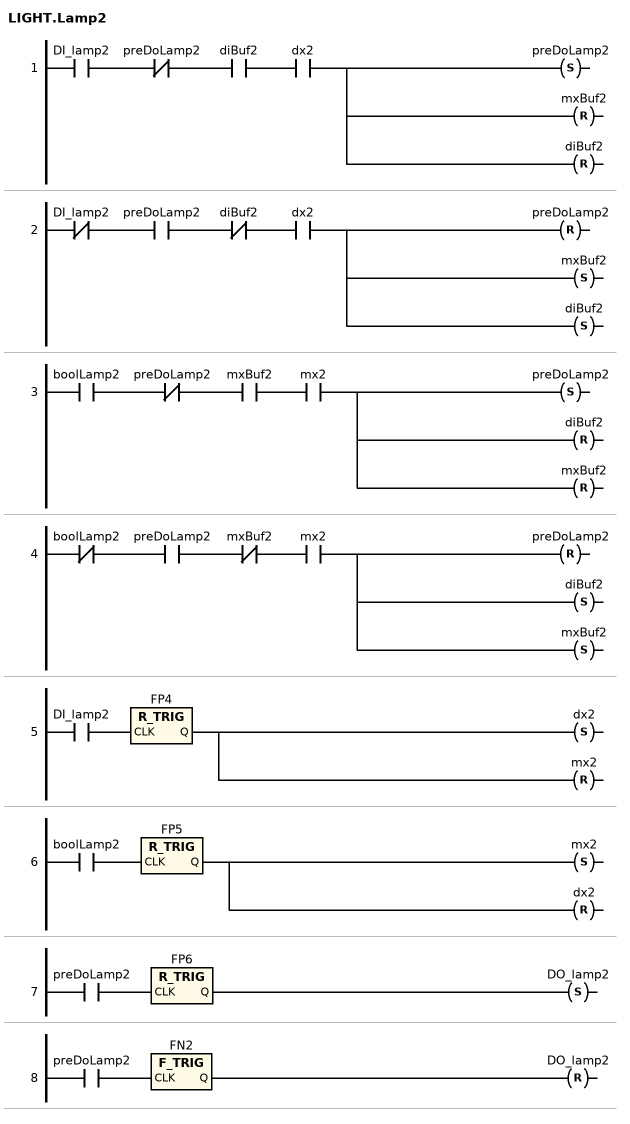
_LD_ (* Ladder Diagram *)
NETWORK 1
	[DI_lamp2] - [/preDoLamp2] - [diBuf2] - [dx2] --- (S preDoLamp2) (R mxBuf2) (R diBuf2)
NETWORK 2
	[/DI_lamp2] - [preDoLamp2] - [/diBuf2] - [dx2] --- (R preDoLamp2) (S mxBuf2) (S diBuf2)
NETWORK 3
	[boolLamp2] - [/preDoLamp2] - [mxBuf2] - [mx2] --- (S preDoLamp2) (R diBuf2) (R mxBuf2)
NETWORK 4
	[/boolLamp2] - [preDoLamp2] - [/mxBuf2] - [mx2] --- (R preDoLamp2) (S diBuf2) (S mxBuf2)
NETWORK 5
	[DI_lamp2] - FP4:R_TRIG(CLK: *) --- (S dx2) (R mx2)
NETWORK 6
	[boolLamp2] - FP5:R_TRIG(CLK: *) --- (S mx2) (R dx2)
NETWORK 7
	[preDoLamp2] - FP6:R_TRIG(CLK: *) --- (S DO_lamp2)
NETWORK 8
	[preDoLamp2] - FN2:F_TRIG(CLK: *) --- (R DO_lamp2)
_END_LD_
(* the same logic as Structured Text *)
(* Network 1 *)
_p5 := DI_lamp2 AND NOT preDoLamp2 AND diBuf2 AND dx2;
IF _p5 THEN preDoLamp2 := TRUE; mxBuf2 := FALSE; diBuf2 := FALSE; END_IF;
(* Network 2 *)
_p6 := NOT DI_lamp2 AND preDoLamp2 AND NOT diBuf2 AND dx2;
IF _p6 THEN preDoLamp2 := FALSE; mxBuf2 := TRUE; diBuf2 := TRUE; END_IF;
(* Network 3 *)
_p7 := boolLamp2 AND NOT preDoLamp2 AND mxBuf2 AND mx2;
IF _p7 THEN preDoLamp2 := TRUE; diBuf2 := FALSE; mxBuf2 := FALSE; END_IF;
(* Network 4 *)
_p8 := NOT boolLamp2 AND preDoLamp2 AND NOT mxBuf2 AND mx2;
IF _p8 THEN preDoLamp2 := FALSE; diBuf2 := TRUE; mxBuf2 := TRUE; END_IF;
(* Network 5 *)
FP4(CLK := DI_lamp2);
IF FP4.Q THEN dx2 := TRUE; mx2 := FALSE; END_IF;
(* Network 6 *)
FP5(CLK := boolLamp2);
IF FP5.Q THEN mx2 := TRUE; dx2 := FALSE; END_IF;
(* Network 7 *)
FP6(CLK := preDoLamp2);
IF FP6.Q THEN DO_lamp2 := TRUE; END_IF;
(* Network 8 *)
FN2(CLK := preDoLamp2);
IF FN2.Q THEN DO_lamp2 := FALSE; END_IF;
END_ACTION
ACTION Lamp3:
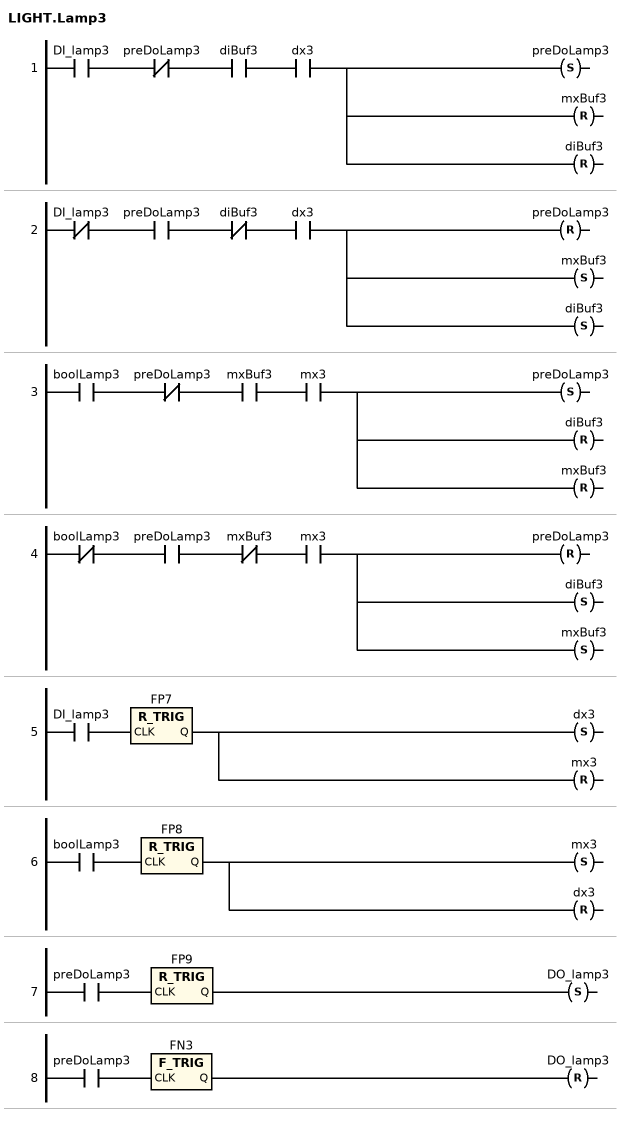
_LD_ (* Ladder Diagram *)
NETWORK 1
	[DI_lamp3] - [/preDoLamp3] - [diBuf3] - [dx3] --- (S preDoLamp3) (R mxBuf3) (R diBuf3)
NETWORK 2
	[/DI_lamp3] - [preDoLamp3] - [/diBuf3] - [dx3] --- (R preDoLamp3) (S mxBuf3) (S diBuf3)
NETWORK 3
	[boolLamp3] - [/preDoLamp3] - [mxBuf3] - [mx3] --- (S preDoLamp3) (R diBuf3) (R mxBuf3)
NETWORK 4
	[/boolLamp3] - [preDoLamp3] - [/mxBuf3] - [mx3] --- (R preDoLamp3) (S diBuf3) (S mxBuf3)
NETWORK 5
	[DI_lamp3] - FP7:R_TRIG(CLK: *) --- (S dx3) (R mx3)
NETWORK 6
	[boolLamp3] - FP8:R_TRIG(CLK: *) --- (S mx3) (R dx3)
NETWORK 7
	[preDoLamp3] - FP9:R_TRIG(CLK: *) --- (S DO_lamp3)
NETWORK 8
	[preDoLamp3] - FN3:F_TRIG(CLK: *) --- (R DO_lamp3)
_END_LD_
(* the same logic as Structured Text *)
(* Network 1 *)
_p9 := DI_lamp3 AND NOT preDoLamp3 AND diBuf3 AND dx3;
IF _p9 THEN preDoLamp3 := TRUE; mxBuf3 := FALSE; diBuf3 := FALSE; END_IF;
(* Network 2 *)
_p10 := NOT DI_lamp3 AND preDoLamp3 AND NOT diBuf3 AND dx3;
IF _p10 THEN preDoLamp3 := FALSE; mxBuf3 := TRUE; diBuf3 := TRUE; END_IF;
(* Network 3 *)
_p11 := boolLamp3 AND NOT preDoLamp3 AND mxBuf3 AND mx3;
IF _p11 THEN preDoLamp3 := TRUE; diBuf3 := FALSE; mxBuf3 := FALSE; END_IF;
(* Network 4 *)
_p12 := NOT boolLamp3 AND preDoLamp3 AND NOT mxBuf3 AND mx3;
IF _p12 THEN preDoLamp3 := FALSE; diBuf3 := TRUE; mxBuf3 := TRUE; END_IF;
(* Network 5 *)
FP7(CLK := DI_lamp3);
IF FP7.Q THEN dx3 := TRUE; mx3 := FALSE; END_IF;
(* Network 6 *)
FP8(CLK := boolLamp3);
IF FP8.Q THEN mx3 := TRUE; dx3 := FALSE; END_IF;
(* Network 7 *)
FP9(CLK := preDoLamp3);
IF FP9.Q THEN DO_lamp3 := TRUE; END_IF;
(* Network 8 *)
FN3(CLK := preDoLamp3);
IF FN3.Q THEN DO_lamp3 := FALSE; END_IF;
END_ACTION
ACTION Schedule:
(* 1 *)
IF ( lamp1OnHH = TimeAndDate.Hour ) AND ( lamp1OnMM = TimeAndDate.Minute ) AND ( TimeAndDate.Second = 0 )
	THEN DO_lamp1 := TRUE;
END_IF;

IF ( lamp1OffHH = TimeAndDate.Hour ) AND ( lamp1OffMM = TimeAndDate.Minute ) AND ( TimeAndDate.Second = 0 )
	THEN DO_lamp1 := FALSE;
END_IF;

(* 2 *)
IF ( lamp2OnHH = TimeAndDate.Hour ) AND ( lamp2OnMM = TimeAndDate.Minute ) AND ( TimeAndDate.Second = 0 )
	THEN DO_lamp2 := TRUE;
END_IF;

IF ( lamp2OffHH = TimeAndDate.Hour ) AND ( lamp2OffMM = TimeAndDate.Minute ) AND ( TimeAndDate.Second = 0 )
	THEN DO_lamp2 := FALSE;
END_IF;

(* 3 *)
IF ( lamp3OnHH = TimeAndDate.Hour ) AND ( lamp3OnMM = TimeAndDate.Minute ) AND ( TimeAndDate.Second = 0 )
	THEN DO_lamp3 := TRUE;
END_IF;

IF ( lamp3OffHH = TimeAndDate.Hour ) AND ( lamp3OffMM = TimeAndDate.Minute ) AND ( TimeAndDate.Second = 0 )
	THEN DO_lamp3 := FALSE;
END_IF;
END_ACTION
ACTION UnpackTime:
(*
	lo,hi : byte
	w : word

	lo := word_to_byte(w)
	hi := word_to_byte(w/256)
	w := 256*hi + lo 
*)
	lamp1OnHH := WORD_TO_BYTE ( lamp1On );
	lamp1OnMM := WORD_TO_BYTE ( lamp1On / 256 );

	lamp1OffHH := WORD_TO_BYTE ( lamp1Off );
	lamp1OffMM := WORD_TO_BYTE ( lamp1Off / 256 );


	lamp2OnHH := WORD_TO_BYTE ( lamp2On );
	lamp2OnMM := WORD_TO_BYTE ( lamp2On / 256 );

	lamp2OffHH := WORD_TO_BYTE ( lamp2Off );
	lamp2OffMM := WORD_TO_BYTE ( lamp2Off / 256 );


	lamp3OnHH := WORD_TO_BYTE ( lamp3On );
	lamp3OnMM := WORD_TO_BYTE ( lamp3On / 256 );

	lamp3OffHH := WORD_TO_BYTE ( lamp3Off );
	lamp3OffMM := WORD_TO_BYTE ( lamp3Off / 256 );
END_ACTION
ACTION WithdrawRetain:
dim1 := dim1_save;
dim2 := dim2_save;
dim3 := dim3_save;

lamp1On := lamp1On_save;
lamp1Off := lamp1Off_save;
lamp2On := lamp2On_save;
lamp2Off := lamp2Off_save;
lamp3On := lamp3On_save;
lamp3Off := lamp3Off_save;
END_ACTION

(* POU DRENAGE, ST *)
PROGRAM DRENAGE
VAR
	NO_FIRST_PASS : BOOL;
	level : REAL;
	top, bottom : REAL;
	auto, manstart : BOOL;
	pumpStart, pumpGo,	pumpStop : BOOL;
	autoStart: BOOL;
	timerGo: BOOL;
	T1: TON;
	T2: TON;
	timerStop: BOOL;
END_VAR
VAR RETAIN
	sens4ma_save, sens20ma_save : WORD;
	top_save, bottom_save : WORD;
	DrenageBITS_save : WORD;
END_VAR
IF NO_FIRST_PASS = FALSE
	THEN WithdrawRetain;
			NO_FIRST_PASS := TRUE;
END_IF;

CheckNewValue;

Calibration;

auto := DrenageBITS.0;
manstart := DrenageBITS.1;
top := WORD_TO_REAL ( dist_top ) / 100;
bottom := WORD_TO_REAL ( dist_bottom ) / 100;

main;

DO_drePump := pumpStart;
dreOUT.0 := pumpStart;

(*----------------------*)

IF DrenageBITS.2
	THEN DO_unknownPump := TRUE;
	ELSE DO_unknownPump := FALSE;
END_IF;

IF DO_unknownPump
	THEN dreOUT.1 := TRUE;
	ELSE dreOUT.1 := FALSE;
END_IF;
END_PROGRAM
ACTION Calibration:
(* Result = n2 + ( Input - n1 ) * ( ( m2 - n2 ) / ( m1 - n1 ) ) *)


	(* panPres := pan4mA / 10  + ( AI_pres - 4 ) * ( ( pan20mA / 10 ) - (  pan4mA / 10 ) ) / 16; *)

(*	wordpres := REAL_TO_INT ( ( pan4mA / 10  + ( AI_pres - 4 ) * ( ( pan20mA / 10 ) - (  pan4mA / 10 ) ) / 16 ) * 100 ); *)

level := sens4ma / 100 + ( AI_02 / 1000 - 4 ) * ( ( sens20ma / 100 ) - ( sens4ma / 100 ) ) / 16;
END_ACTION
ACTION CheckNewValue:
IF DrenageBITS_save <> DrenageBITS
	THEN DrenageBITS_save := DrenageBITS;
END_IF;

IF top_save <> dist_top
	THEN top_save := dist_top;
END_IF;

IF bottom_save <> dist_bottom
	THEN bottom_save := dist_bottom;
END_IF;

IF sens4ma_save <> sens4ma
	THEN sens4ma_save := sens4ma;
END_IF;

IF sens20ma_save <> sens20ma
	THEN sens20ma_save := sens20ma;
END_IF;
END_ACTION
ACTION main:
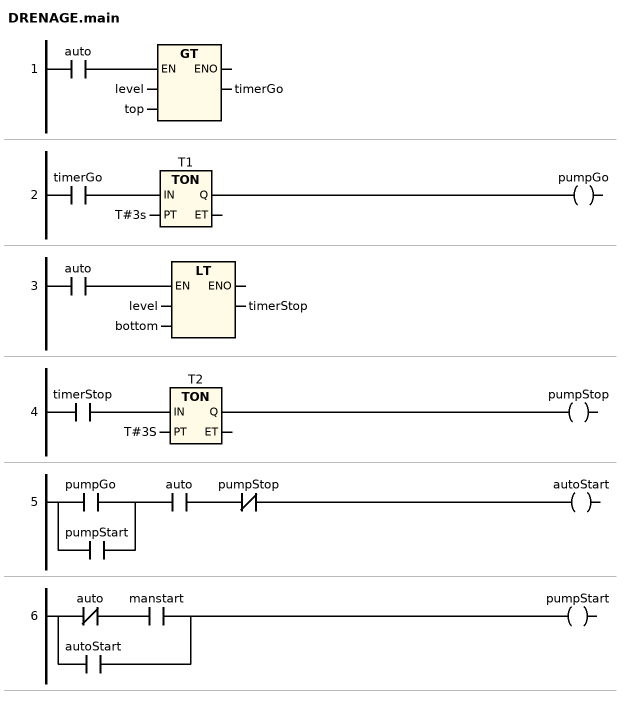
_LD_ (* Ladder Diagram *)
NETWORK 1
	[auto]
		EN --- GT(level, top) => timerGo
NETWORK 2
	[timerGo] - T1:TON(IN: *, PT: T#3s) --- (pumpGo)
NETWORK 3
	[auto]
		EN --- LT(level, bottom) => timerStop
NETWORK 4
	[timerStop] - T2:TON(IN: *, PT: T#3S) --- (pumpStop)
NETWORK 5
	{ [pumpGo] | [pumpStart] } - [auto] - [/pumpStop] --- (autoStart)
NETWORK 6
	{ [/auto] - [manstart] | [autoStart] } --- (pumpStart)
_END_LD_
(* the same logic as Structured Text *)
(* Network 1 *)
IF auto THEN
	timerGo := level > top;
END_IF;
(* Network 2 *)
T1(IN := timerGo, PT := T#3s);
pumpGo := T1.Q;
(* Network 3 *)
IF auto THEN
	timerStop := level < bottom;
END_IF;
(* Network 4 *)
T2(IN := timerStop, PT := T#3S);
pumpStop := T2.Q;
(* Network 5 *)
autoStart := (pumpGo OR pumpStart) AND auto AND NOT pumpStop;
(* Network 6 *)
pumpStart := NOT auto AND manstart OR autoStart;
END_ACTION
ACTION WithdrawRetain:
dist_top := top_save / 100;
dist_bottom := bottom_save / 100;

DrenageBITS := DrenageBITS_save;

sens4ma := sens4ma_save;
sens20ma := sens20ma_save;
END_ACTION

(* POU SMS, ST *)
PROGRAM SMS
VAR
	Com		: OpenPort;
	cfg		       : FB_SMS_CFG;
	sms		:FB_SMS_SR;
	cfg_ok		: BOOL := FALSE;
	sendSMS  : BOOL := FALSE;
	ready		: BOOL;
	DevNum	: WORD := 0;
	openModemPort : BOOL := FALSE;
	port_ok      : BOOL := FALSE;
	errCode     : BYTE;
	errBool      : BOOL;

	sendText   : STRING(70);
	sended     : BOOL;

	senderErrCode : BYTE;
	timeOut : TON;

	lock1, lock2, lock3, lock4 : BOOL := FALSE;
END_VAR
Inputs;

IF SMS_ID > 0 THEN
	Select;
	openModemPort := TRUE;
	sendSMS := TRUE;
ELSE
	openModemPort := FALSE;
	sendSMS := FALSE;
END_IF;

Configure;

IF ( cfg_ok=TRUE ) AND ( errBool=FALSE ) THEN

	ready := TRUE;
ELSE
	ready := FALSE;
END_IF;

Send;

IF sended THEN
	SMS_ID := 0;
	sendSMS := FALSE;
END_IF;

Timeout;
END_PROGRAM
ACTION Configure:
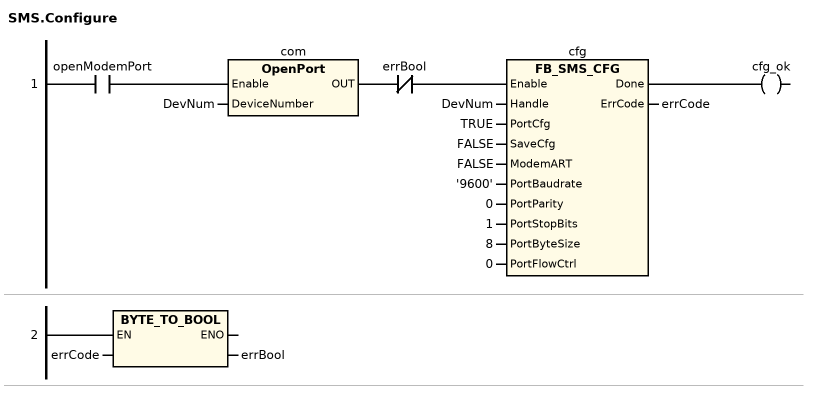
_LD_ (* Ladder Diagram *)
NETWORK 1
	[openModemPort] - com:OpenPort(Enable: *, DeviceNumber: DevNum) - [/errBool] - cfg:FB_SMS_CFG(Enable: *, Handle: DevNum, PortCfg: TRUE, SaveCfg: FALSE, ModemART: FALSE, PortBaudrate: '9600', PortParity: 0, PortStopBits: 1, PortByteSize: 8, PortFlowCtrl: 0, ErrCode => errCode) --- (cfg_ok)
NETWORK 2
	*
		EN --- BYTE_TO_BOOL(errCode) => errBool
_END_LD_
(* the same logic as Structured Text *)
(* Network 1 *)
com(Enable := openModemPort, DeviceNumber := DevNum);
cfg(Enable := com.OUT AND NOT errBool, Handle := DevNum, PortCfg := TRUE, SaveCfg := FALSE, ModemART := FALSE, PortBaudrate := '9600', PortParity := 0, PortStopBits := 1, PortByteSize := 8, PortFlowCtrl := 0);
errCode := cfg.ErrCode;
cfg_ok := cfg.Done;
(* Network 2 *)
errBool := BYTE_TO_BOOL(errCode);
END_ACTION
ACTION Inputs:
IF SMS_ID = 0 THEN
	IF DI_powerSupply AND lock1=FALSE THEN
		SMS_ID := 1;
		lock1 := TRUE;
	END_IF;
	IF DI_signal1 AND lock2=FALSE THEN
		SMS_ID := 2;
		lock2 := TRUE;
	END_IF;
	IF DI_signal2 AND lock3=FALSE THEN
		SMS_ID := 4;
		lock3 := TRUE;
	END_IF;
	IF DI_fireSignal AND lock4=FALSE THEN
		SMS_ID := 8;
		lock4 := TRUE;
	END_IF;
END_IF;

IF DI_powerSupply=FALSE THEN
	lock1 := FALSE;
END_IF;
IF DI_signal1=FALSE THEN
	lock2 := FALSE;
END_IF;
IF DI_signal2=FALSE THEN
	lock3 := FALSE;
END_IF;
IF DI_fireSignal=FALSE THEN
	lock4 := FALSE;
END_IF;
END_ACTION
ACTION Select:
IF SMS_ID.0 THEN
	sendText := 'Блок питания';
END_IF;

IF SMS_ID.1 THEN
	sendText := 'Извещатель охранный';
END_IF;

IF SMS_ID.2 THEN
	sendText := 'Извещатель объёмный';
END_IF;

IF SMS_ID.3 THEN
	sendText := 'Извещатель пожарный дымовой';
END_IF;
END_ACTION
ACTION Send:
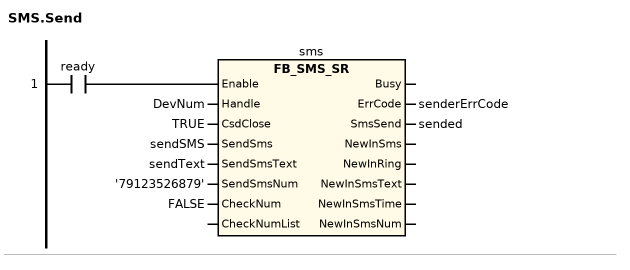
_LD_ (* Ladder Diagram *)
NETWORK 1
	[ready] - sms:FB_SMS_SR(Enable: *, Handle: DevNum, CsdClose: TRUE, SendSms: sendSMS, SendSmsText: sendText, SendSmsNum: '79123526879', CheckNum: FALSE, CheckNumList: , ErrCode => senderErrCode, SmsSend => sended)
_END_LD_
END_ACTION
ACTION Timeout:
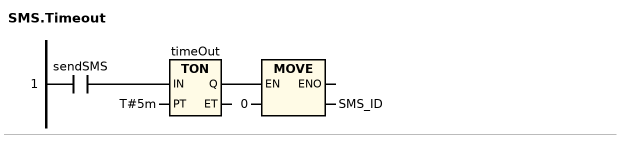
_LD_ (* Ladder Diagram *)
NETWORK 1
	[sendSMS] - timeOut:TON(IN: *, PT: T#5m)
		EN --- MOVE(0) => SMS_ID
_END_LD_
(* the same logic as Structured Text *)
(* Network 1 *)
timeOut(IN := sendSMS, PT := T#5m);
IF timeOut.Q THEN
	SMS_ID := 0;
END_IF;
END_ACTION
